LIN {X 0,Y 291.334,Z 480.193,A -85,B 0,C 180,E1 -16780.643,E2 -16780.643} C_VEL
LIN {X 0,Y 291.294,Z 480.201,A -85,B 0,C 180,E1 -16784.402,E2 -16784.402} C_VEL
LIN {X 0,Y 291.33,Z 480.196,A -85,B 0,C 180,E1 -16788.405,E2 -16788.405} C_VEL
LIN {X 0,Y 291.368,Z 480.187,A -85,B 0,C 180,E1 -16791.161,E2 -16791.161} C_VEL
LIN {X 0,Y 291.389,Z 480.187,A -85,B 0,C 180,E1 -16794.63,E2 -16794.63} C_VEL
LIN {X 0,Y 291.377,Z 480.19,A -85,B 0,C 180,E1 -16797.951,E2 -16797.951} C_VEL
LIN {X 0,Y 291.386,Z 480.185,A -85,B 0,C 180,E1 -16801.159,E2 -16801.159} C_VEL
LIN {X 0,Y 291.422,Z 480.185,A -85,B 0,C 180,E1 -16804.272,E2 -16804.272} C_VEL
LIN {X 0,Y 291.386,Z 480.185,A -85,B 0,C 180,E1 -16807.3,E2 -16807.3} C_VEL
LIN {X 0,Y 291.463,Z 480.18,A -85,B 0,C 180,E1 -16810.27,E2 -16810.27} C_VEL
LIN {X 0,Y 291.56,Z 480.165,A -85,B 0,C 180,E1 -16814.624,E2 -16814.624} C_VEL
LIN {X 0,Y 291.542,Z 480.166,A -85,B 0,C 180,E1 -16818.881,E2 -16818.881} C_VEL
LIN {X 0,Y 291.714,Z 480.147,A -85,B 0,C 180,E1 -16821.689,E2 -16821.689} C_VEL
LIN {X 0,Y 291.635,Z 480.156,A -85,B 0,C 180,E1 -16824.468,E2 -16824.468} C_VEL
LIN {X 0,Y 291.893,Z 480.123,A -85,B 0,C 180,E1 -16828.62,E2 -16828.62} C_VEL
LIN {X 0,Y 291.893,Z 480.123,A -85,B 0,C 180,E1 -16831.38,E2 -16831.38} C_VEL
LIN {X 0,Y 291.616,Z 480.158,A -85,B 0,C 180,E1 -16835.532,E2 -16835.532} C_VEL
LIN {X 0,Y 291.678,Z 480.149,A -85,B 0,C 180,E1 -16838.919,E2 -16838.919} C_VEL
LIN {X 0,Y 291.525,Z 480.168,A -85,B 0,C 180,E1 -16842.531,E2 -16842.531} C_VEL
LIN {X 0,Y 291.56,Z 480.165,A -85,B 0,C 180,E1 -16845.376,E2 -16845.376} C_VEL
LIN {X 0,Y 291.455,Z 480.182,A -85,B 0,C 180,E1 -16849.875,E2 -16849.875} C_VEL
LIN {X 0,Y 291.403,Z 480.186,A -85,B 0,C 180,E1 -16854.205,E2 -16854.205} C_VEL
LIN {X 0,Y 291.424,Z 480.182,A -85,B 0,C 180,E1 -16857.272,E2 -16857.272} C_VEL
LIN {X 0,Y 291.338,Z 480.191,A -85,B 0,C 180,E1 -16860.437,E2 -16860.437} C_VEL
LIN {X 0,Y 291.349,Z 480.194,A -85,B 0,C 180,E1 -16863.698,E2 -16863.698} C_VEL
LIN {X 0,Y 291.398,Z 480.185,A -85,B 0,C 180,E1 -16867.259,E2 -16867.259} C_VEL
LIN {X 0,Y 291.338,Z 480.191,A -85,B 0,C 180,E1 -16870.642,E2 -16870.642} C_VEL
LIN {X 0,Y 291.293,Z 480.198,A -85,B 0,C 180,E1 -16874.402,E2 -16874.402} C_VEL
LIN {X 0,Y 291.329,Z 480.192,A -85,B 0,C 180,E1 -16878.404,E2 -16878.404} C_VEL
LIN {X 0,Y 291.347,Z 480.192,A -85,B 0,C 180,E1 -16881.157,E2 -16881.157} C_VEL
LIN {X 0,Y 291.375,Z 480.187,A -85,B 0,C 180,E1 -16882.914,E2 -16882.914} C_VEL
LIN {X 0,Y 291.126,Z 480.218,A -85,B 0,C 180,E1 -16886.272,E2 -16886.272} C_VEL
LIN {X 0,Y 290.796,Z 480.263,A -85,B 0,C 180,E1 -16889.5,E2 -16889.5} C_VEL
LIN {X 0,Y 290.411,Z 480.307,A -85,B 0,C 180,E1 -16892.625,E2 -16892.625} C_VEL
LIN {X 0,Y 289.943,Z 480.417,A -85,B 0,C 180,E1 -16896.236,E2 -16896.236} C_VEL
LIN {X 0,Y 289.946,Z 482.927,A -85,B 0,C 180,E1 -16898.679,E2 -16898.679} C_VEL
LIN {X 0,Y 292.691,Z 498.006,A -85,B 0,C 180,E1 -16899.711,E2 -16899.711} C_VEL
LIN {X 0,Y 295.355,Z 512.188,A -85,B 0,C 180,E1 -16900.992,E2 -16900.992} C_VEL
LIN {X 0,Y 295.583,Z 516.745,A -85,B 0,C 180,E1 -16901.457,E2 -16901.457} C_VEL
LIN {X 0,Y 294.542,Z 528.4,A -85,B 0,C 180,E1 -16902.788,E2 -16902.788} C_VEL
LIN {X 0,Y 293.546,Z 538.437,A -85,B 0,C 180,E1 -16904.196,E2 -16904.196} C_VEL
LIN {X 0,Y 292.641,Z 547.665,A -85,B 0,C 180,E1 -16905.749,E2 -16905.749} C_VEL
LIN {X 0,Y 291.737,Z 556.266,A -85,B 0,C 180,E1 -16907.478,E2 -16907.478} C_VEL
LIN {X 0,Y 290.974,Z 564.767,A -85,B 0,C 180,E1 -16909.563,E2 -16909.563} C_VEL
LIN {X 0,Y 290.377,Z 571.664,A -85,B 0,C 180,E1 -16911.65,E2 -16911.65} C_VEL
LIN {X 0,Y 290.067,Z 576.41,A -85,B 0,C 180,E1 -16913.408,E2 -16913.408} C_VEL
LIN {X 0,Y 289.833,Z 581.565,A -85,B 0,C 180,E1 -16915.828,E2 -16915.828} C_VEL
LIN {X 0,Y 289.714,Z 583.883,A -85,B 0,C 180,E1 -16917.219,E2 -16917.219} C_VEL
LIN {X 0,Y 289.64,Z 585.506,A -85,B 0,C 180,E1 -16918.442,E2 -16918.442} C_VEL
LIN {X 0,Y 289.01,Z 586.88,A -85,B 0,C 180,E1 -16919.573,E2 -16919.573} C_VEL
LIN {X 0,Y 286.338,Z 588.547,A -85,B 0,C 180,E1 -16921.444,E2 -16921.444} C_VEL
LIN {X 0,Y 284.137,Z 589.296,A -85,B 0,C 180,E1 -16922.979,E2 -16922.979} C_VEL
LIN {X 0,Y 283.277,Z 589.509,A -85,B 0,C 180,E1 -16924.167,E2 -16924.167} C_VEL
LIN {X 0,Y 283.251,Z 589.501,A -85,B 0,C 180,E1 -16924.568,E2 -16924.568} C_VEL
LIN {X 0,Y 283.807,Z 588.988,A -85,B 0,C 180,E1 -16927.112,E2 -16927.112} C_VEL
LIN {X 0,Y 285.067,Z 587.261,A -85,B 0,C 180,E1 -16929.544,E2 -16929.544} C_VEL
LIN {X 0,Y 286.508,Z 584.256,A -85,B 0,C 180,E1 -16932.034,E2 -16932.034} C_VEL
LIN {X 0,Y 288.806,Z 579.257,A -85,B 0,C 180,E1 -16934.804,E2 -16934.804} C_VEL
LIN {X 0,Y 290.955,Z 574.336,A -85,B 0,C 180,E1 -16936.849,E2 -16936.849} C_VEL
LIN {X 0,Y 293.872,Z 567.073,A -85,B 0,C 180,E1 -16939.198,E2 -16939.198} C_VEL
LIN {X 0,Y 296.873,Z 559.452,A -85,B 0,C 180,E1 -16941.163,E2 -16941.163} C_VEL
LIN {X 0,Y 300.223,Z 550.179,A -85,B 0,C 180,E1 -16943.085,E2 -16943.085} C_VEL
LIN {X 0,Y 303.614,Z 539.794,A -85,B 0,C 180,E1 -16944.831,E2 -16944.831} C_VEL
LIN {X 0,Y 304.404,Z 537.308,A -85,B 0,C 180,E1 -16945.191,E2 -16945.191} C_VEL
LIN {X 0,Y 304.646,Z 535.637,A -85,B 0,C 180,E1 -16945.489,E2 -16945.489} C_VEL
LIN {X 0,Y 303.451,Z 527.808,A -85,B 0,C 180,E1 -16947.303,E2 -16947.303} C_VEL
LIN {X 0,Y 301.243,Z 520.052,A -85,B 0,C 180,E1 -16949.336,E2 -16949.336} C_VEL
LIN {X 0,Y 298.599,Z 513.072,A -85,B 0,C 180,E1 -16951.459,E2 -16951.459} C_VEL
LIN {X 0,Y 296.624,Z 508.611,A -85,B 0,C 180,E1 -16953.021,E2 -16953.021} C_VEL
LIN {X 0,Y 294.159,Z 504.223,A -85,B 0,C 180,E1 -16954.988,E2 -16954.988} C_VEL
LIN {X 0,Y 291.916,Z 500.866,A -85,B 0,C 180,E1 -16957.005,E2 -16957.005} C_VEL
LIN {X 0,Y 291.673,Z 500.148,A -85,B 0,C 180,E1 -16957.33,E2 -16957.33} C_VEL
LIN {X 0,Y 288.682,Z 497.206,A -85,B 0,C 180,E1 -16961.096,E2 -16961.096} C_VEL
LIN {X 0,Y 288.16,Z 496.183,A -85,B 0,C 180,E1 -16963.31,E2 -16963.31} C_VEL
LIN {X 0,Y 288.331,Z 496.661,A -85,B 0,C 180,E1 -16965.019,E2 -16965.019} C_VEL
LIN {X 0,Y 288.629,Z 498.198,A -85,B 0,C 180,E1 -16967.855,E2 -16967.855} C_VEL
LIN {X 0,Y 290.515,Z 502.885,A -85,B 0,C 180,E1 -16971.025,E2 -16971.025} C_VEL
LIN {X 0,Y 292.089,Z 505.556,A -85,B 0,C 180,E1 -16972.563,E2 -16972.563} C_VEL
LIN {X 0,Y 294.502,Z 513.126,A -85,B 0,C 180,E1 -16975.059,E2 -16975.059} C_VEL
LIN {X 0,Y 296.539,Z 520.344,A -85,B 0,C 180,E1 -16976.968,E2 -16976.968} C_VEL
LIN {X 0,Y 297.747,Z 527.635,A -85,B 0,C 180,E1 -16978.485,E2 -16978.485} C_VEL
LIN {X 0,Y 299.033,Z 539.159,A -85,B 0,C 180,E1 -16980.658,E2 -16980.658} C_VEL
LIN {X 0,Y 299.343,Z 551.45,A -85,B 0,C 180,E1 -16982.829,E2 -16982.829} C_VEL
LIN {X 0,Y 298.611,Z 562.364,A -85,B 0,C 180,E1 -16984.739,E2 -16984.739} C_VEL
LIN {X 0,Y 296.615,Z 572.882,A -85,B 0,C 180,E1 -16986.617,E2 -16986.617} C_VEL
LIN {X 0,Y 293.295,Z 582.962,A -85,B 0,C 180,E1 -16988.566,E2 -16988.566} C_VEL
LIN {X 0,Y 290.399,Z 591.537,A -85,B 0,C 180,E1 -16990.609,E2 -16990.609} C_VEL
LIN {X 0,Y 288.013,Z 598.477,A -85,B 0,C 180,E1 -16992.607,E2 -16992.607} C_VEL
LIN {X 0,Y 285.907,Z 605.175,A -85,B 0,C 180,E1 -16995.042,E2 -16995.042} C_VEL
LIN {X 0,Y 284.328,Z 609.813,A -85,B 0,C 180,E1 -16997.146,E2 -16997.146} C_VEL
LIN {X 0,Y 283.152,Z 614.446,A -85,B 0,C 180,E1 -16999.994,E2 -16999.994} C_VEL
LIN {X 0,Y 282.803,Z 616.163,A -85,B 0,C 180,E1 -17001.425,E2 -17001.425} C_VEL
LIN {X 0,Y 282.522,Z 618.348,A -85,B 0,C 180,E1 -17004.289,E2 -17004.289} C_VEL
LIN {X 0,Y 282.52,Z 618.859,A -85,B 0,C 180,E1 -17005.72,E2 -17005.72} C_VEL
LIN {X 0,Y 282.582,Z 618.969,A -85,B 0,C 180,E1 -17007.149,E2 -17007.149} C_VEL
LIN {X 0,Y 282.866,Z 618.592,A -85,B 0,C 180,E1 -17008.932,E2 -17008.932} C_VEL
LIN {X 0,Y 282.885,Z 619.433,A -85,B 0,C 180,E1 -17010,E2 -17010} C_VEL
LIN {X 0,Y 282.703,Z 620.169,A -85,B 0,C 180,E1 -17011.425,E2 -17011.425} C_VEL
LIN {X 0,Y 282.498,Z 620.489,A -85,B 0,C 180,E1 -17012.852,E2 -17012.852} C_VEL
LIN {X 0,Y 282.442,Z 619.945,A -85,B 0,C 180,E1 -17015.546,E2 -17015.546} C_VEL
LIN {X 0,Y 282.549,Z 618.968,A -85,B 0,C 180,E1 -17017.144,E2 -17017.144} C_VEL
LIN {X 0,Y 282.796,Z 617.689,A -85,B 0,C 180,E1 -17018.575,E2 -17018.575} C_VEL
LIN {X 0,Y 283.705,Z 613.888,A -85,B 0,C 180,E1 -17021.43,E2 -17021.43} C_VEL
LIN {X 0,Y 284.793,Z 609.991,A -85,B 0,C 180,E1 -17023.558,E2 -17023.558} C_VEL
LIN {X 0,Y 286.466,Z 605.074,A -85,B 0,C 180,E1 -17025.656,E2 -17025.656} C_VEL
LIN {X 0,Y 289.04,Z 596.909,A -85,B 0,C 180,E1 -17028.427,E2 -17028.427} C_VEL
LIN {X 0,Y 292.268,Z 587.863,A -85,B 0,C 180,E1 -17030.774,E2 -17030.774} C_VEL
LIN {X 0,Y 295.55,Z 578.572,A -85,B 0,C 180,E1 -17032.732,E2 -17032.732} C_VEL
LIN {X 0,Y 297.766,Z 571.418,A -85,B 0,C 180,E1 -17034.025,E2 -17034.025} C_VEL
LIN {X 0,Y 299.353,Z 562.829,A -85,B 0,C 180,E1 -17035.534,E2 -17035.534} C_VEL
LIN {X 0,Y 299.795,Z 553.607,A -85,B 0,C 180,E1 -17037.202,E2 -17037.202} C_VEL
LIN {X 0,Y 299.141,Z 543.023,A -85,B 0,C 180,E1 -17039.207,E2 -17039.207} C_VEL
LIN {X 0,Y 297.549,Z 532.972,A -85,B 0,C 180,E1 -17041.308,E2 -17041.308} C_VEL
LIN {X 0,Y 295.334,Z 523.354,A -85,B 0,C 180,E1 -17043.603,E2 -17043.603} C_VEL
LIN {X 0,Y 293.444,Z 516.852,A -85,B 0,C 180,E1 -17045.482,E2 -17045.482} C_VEL
LIN {X 0,Y 292.016,Z 512.481,A -85,B 0,C 180,E1 -17046.99,E2 -17046.99} C_VEL
LIN {X 0,Y 291.808,Z 511.167,A -85,B 0,C 180,E1 -17047.365,E2 -17047.365} C_VEL
LIN {X 0,Y 288.758,Z 504.957,A -85,B 0,C 180,E1 -17051.083,E2 -17051.083} C_VEL
LIN {X 0,Y 288.003,Z 501.761,A -85,B 0,C 180,E1 -17053.544,E2 -17053.544} C_VEL
LIN {X 0,Y 287.807,Z 500.618,A -85,B 0,C 180,E1 -17055.975,E2 -17055.975} C_VEL
LIN {X 0,Y 288.439,Z 501.626,A -85,B 0,C 180,E1 -17059.055,E2 -17059.055} C_VEL
LIN {X 0,Y 291.413,Z 503.824,A -85,B 0,C 180,E1 -17062.737,E2 -17062.737} C_VEL
LIN {X 0,Y 292.328,Z 505.916,A -85,B 0,C 180,E1 -17063.863,E2 -17063.863} C_VEL
LIN {X 0,Y 293.661,Z 507.267,A -85,B 0,C 180,E1 -17064.944,E2 -17064.944} C_VEL
LIN {X 0,Y 296.553,Z 512.135,A -85,B 0,C 180,E1 -17067.281,E2 -17067.281} C_VEL
LIN {X 0,Y 300.148,Z 519.88,A -85,B 0,C 180,E1 -17070.039,E2 -17070.039} C_VEL
LIN {X 0,Y 302.846,Z 527.891,A -85,B 0,C 180,E1 -17072.346,E2 -17072.346} C_VEL
LIN {X 0,Y 304.613,Z 536.548,A -85,B 0,C 180,E1 -17074.514,E2 -17074.514} C_VEL
LIN {X 0,Y 304.698,Z 537.826,A -85,B 0,C 180,E1 -17074.798,E2 -17074.798} C_VEL
LIN {X 0,Y 301.105,Z 548.999,A -85,B 0,C 180,E1 -17076.622,E2 -17076.622} C_VEL
LIN {X 0,Y 297.665,Z 558.567,A -85,B 0,C 180,E1 -17078.533,E2 -17078.533} C_VEL
LIN {X 0,Y 294.039,Z 567.574,A -85,B 0,C 180,E1 -17080.814,E2 -17080.814} C_VEL
LIN {X 0,Y 291.091,Z 574.794,A -85,B 0,C 180,E1 -17083.159,E2 -17083.159} C_VEL
LIN {X 0,Y 288.974,Z 579.689,A -85,B 0,C 180,E1 -17085.205,E2 -17085.205} C_VEL
LIN {X 0,Y 286.607,Z 584.705,A -85,B 0,C 180,E1 -17087.97,E2 -17087.97} C_VEL
LIN {X 0,Y 285.258,Z 587.491,A -85,B 0,C 180,E1 -17090.231,E2 -17090.231} C_VEL
LIN {X 0,Y 283.867,Z 589.466,A -85,B 0,C 180,E1 -17092.889,E2 -17092.889} C_VEL
LIN {X 0,Y 283.578,Z 589.924,A -85,B 0,C 180,E1 -17094.311,E2 -17094.311} C_VEL
LIN {X 0,Y 283.299,Z 590.016,A -85,B 0,C 180,E1 -17095.732,E2 -17095.732} C_VEL
LIN {X 0,Y 282.979,Z 589.737,A -85,B 0,C 180,E1 -17097.153,E2 -17097.153} C_VEL
LIN {X 0,Y 282.754,Z 589.038,A -85,B 0,C 180,E1 -17098.576,E2 -17098.576} C_VEL
LIN {X 0,Y 282.586,Z 586.427,A -85,B 0,C 180,E1 -17101.425,E2 -17101.425} C_VEL
LIN {X 0,Y 282.709,Z 583.358,A -85,B 0,C 180,E1 -17103.564,E2 -17103.564} C_VEL
LIN {X 0,Y 282.844,Z 579.26,A -85,B 0,C 180,E1 -17105.704,E2 -17105.704} C_VEL
LIN {X 0,Y 283.281,Z 573.055,A -85,B 0,C 180,E1 -17108.202,E2 -17108.202} C_VEL
LIN {X 0,Y 283.949,Z 565.036,A -85,B 0,C 180,E1 -17110.698,E2 -17110.698} C_VEL
LIN {X 0,Y 284.75,Z 556.478,A -85,B 0,C 180,E1 -17112.835,E2 -17112.835} C_VEL
LIN {X 0,Y 285.914,Z 545.866,A -85,B 0,C 180,E1 -17114.958,E2 -17114.958} C_VEL
LIN {X 0,Y 287.022,Z 536.197,A -85,B 0,C 180,E1 -17116.538,E2 -17116.538} C_VEL
LIN {X 0,Y 287.925,Z 525.259,A -85,B 0,C 180,E1 -17118.012,E2 -17118.012} C_VEL
LIN {X 0,Y 288.683,Z 516.455,A -85,B 0,C 180,E1 -17119.003,E2 -17119.003} C_VEL
LIN {X 0,Y 288.131,Z 511.699,A -85,B 0,C 180,E1 -17119.504,E2 -17119.504} C_VEL
LIN {X 0,Y 285.556,Z 498.301,A -85,B 0,C 180,E1 -17120.732,E2 -17120.732} C_VEL
LIN {X 0,Y 282.979,Z 484.536,A -85,B 0,C 180,E1 -17121.705,E2 -17121.705} C_VEL
LIN {X 0,Y 282.92,Z 484.131,A -85,B 0,C 180,E1 -17121.756,E2 -17121.756} C_VEL
LIN {X 0,Y 283.028,Z 481.339,A -85,B 0,C 180,E1 -17124.97,E2 -17124.97} C_VEL
LIN {X 0,Y 283.396,Z 481.187,A -85,B 0,C 180,E1 -17128.112,E2 -17128.112} C_VEL
LIN {X 0,Y 283.732,Z 481.139,A -85,B 0,C 180,E1 -17131.344,E2 -17131.344} C_VEL
LIN {X 0,Y 284.129,Z 481.09,A -85,B 0,C 180,E1 -17135.287,E2 -17135.287} C_VEL
LIN {X 0,Y 284.269,Z 481.077,A -85,B 0,C 180,E1 -17138.176,E2 -17138.176} C_VEL
LIN {X 0,Y 284.275,Z 481.072,A -85,B 0,C 180,E1 -17141.876,E2 -17141.876} C_VEL
LIN {X 0,Y 284.259,Z 481.078,A -85,B 0,C 180,E1 -17146.19,E2 -17146.19} C_VEL
LIN {X 0,Y 284.31,Z 481.07,A -85,B 0,C 180,E1 -17150.024,E2 -17150.024} C_VEL
LIN {X 0,Y 284.354,Z 481.063,A -85,B 0,C 180,E1 -17153.617,E2 -17153.617} C_VEL
LIN {X 0,Y 284.312,Z 481.067,A -85,B 0,C 180,E1 -17157.19,E2 -17157.19} C_VEL
LIN {X 0,Y 284.363,Z 481.064,A -85,B 0,C 180,E1 -17160.376,E2 -17160.376} C_VEL
LIN {X 0,Y 284.382,Z 481.059,A -85,B 0,C 180,E1 -17163.587,E2 -17163.587} C_VEL
LIN {X 0,Y 284.371,Z 481.06,A -85,B 0,C 180,E1 -17166.707,E2 -17166.707} C_VEL
LIN {X 0,Y 284.408,Z 481.055,A -85,B 0,C 180,E1 -17171.262,E2 -17171.262} C_VEL
LIN {X 0,Y 284.497,Z 481.046,A -85,B 0,C 180,E1 -17174.459,E2 -17174.459} C_VEL
LIN {X 0,Y 284.493,Z 481.045,A -85,B 0,C 180,E1 -17178.602,E2 -17178.602} C_VEL
LIN {X 0,Y 284.664,Z 481.024,A -85,B 0,C 180,E1 -17181.481,E2 -17181.481} C_VEL
LIN {X 0,Y 284.606,Z 481.032,A -85,B 0,C 180,E1 -17184.331,E2 -17184.331} C_VEL
LIN {X 0,Y 284.859,Z 481,A -85,B 0,C 180,E1 -17188.586,E2 -17188.586} C_VEL
LIN {X 0,Y 284.859,Z 481,A -85,B 0,C 180,E1 -17191.414,E2 -17191.414} C_VEL
LIN {X 0,Y 284.658,Z 481.024,A -85,B 0,C 180,E1 -17197.091,E2 -17197.091} C_VEL
LIN {X 0,Y 284.522,Z 481.046,A -85,B 0,C 180,E1 -17199.957,E2 -17199.957} C_VEL
LIN {X 0,Y 284.486,Z 481.047,A -85,B 0,C 180,E1 -17204.303,E2 -17204.303} C_VEL
LIN {X 0,Y 284.43,Z 481.053,A -85,B 0,C 180,E1 -17207.248,E2 -17207.248} C_VEL
LIN {X 0,Y 284.382,Z 481.06,A -85,B 0,C 180,E1 -17210.242,E2 -17210.242} C_VEL
LIN {X 0,Y 284.371,Z 481.064,A -85,B 0,C 180,E1 -17213.874,E2 -17213.874} C_VEL
LIN {X 0,Y 284.399,Z 481.057,A -85,B 0,C 180,E1 -17217.173,E2 -17217.173} C_VEL
LIN {X 0,Y 284.298,Z 481.068,A -85,B 0,C 180,E1 -17221.274,E2 -17221.274} C_VEL
LIN {X 0,Y 284.366,Z 481.062,A -85,B 0,C 180,E1 -17225.354,E2 -17225.354} C_VEL
LIN {X 0,Y 284.327,Z 481.066,A -85,B 0,C 180,E1 -17228.167,E2 -17228.167} C_VEL
LIN {X 0,Y 284.273,Z 481.074,A -85,B 0,C 180,E1 -17232.124,E2 -17232.124} C_VEL
LIN {X 0,Y 284.258,Z 481.075,A -85,B 0,C 180,E1 -17236.189,E2 -17236.189} C_VEL
LIN {X 0,Y 284.309,Z 481.07,A -85,B 0,C 180,E1 -17240.024,E2 -17240.024} C_VEL
LIN {X 0,Y 284.254,Z 481.079,A -85,B 0,C 180,E1 -17243.602,E2 -17243.602} C_VEL
LIN {X 0,Y 283.996,Z 481.107,A -85,B 0,C 180,E1 -17247.288,E2 -17247.288} C_VEL
LIN {X 0,Y 283.674,Z 481.147,A -85,B 0,C 180,E1 -17250.297,E2 -17250.297} C_VEL
LIN {X 0,Y 283.27,Z 481.2,A -85,B 0,C 180,E1 -17253.475,E2 -17253.475} C_VEL
LIN {X 0,Y 282.87,Z 481.398,A -85,B 0,C 180,E1 -17256.576,E2 -17256.576} C_VEL
LIN {X 0,Y 282.863,Z 483.281,A -85,B 0,C 180,E1 -17258.43,E2 -17258.43} C_VEL
LIN {X 0,Y 285.601,Z 498.484,A -85,B 0,C 180,E1 -17259.494,E2 -17259.494} C_VEL
LIN {X 0,Y 288.16,Z 512.297,A -85,B 0,C 180,E1 -17260.776,E2 -17260.776} C_VEL
LIN {X 0,Y 288.606,Z 516.076,A -85,B 0,C 180,E1 -17261.176,E2 -17261.176} C_VEL
LIN {X 0,Y 287.539,Z 528.127,A -85,B 0,C 180,E1 -17262.561,E2 -17262.561} C_VEL
LIN {X 0,Y 286.543,Z 538.135,A -85,B 0,C 180,E1 -17263.982,E2 -17263.982} C_VEL
LIN {X 0,Y 285.508,Z 548.416,A -85,B 0,C 180,E1 -17265.749,E2 -17265.749} C_VEL
LIN {X 0,Y 284.62,Z 556.944,A -85,B 0,C 180,E1 -17267.522,E2 -17267.522} C_VEL
LIN {X 0,Y 283.836,Z 565.352,A -85,B 0,C 180,E1 -17269.658,E2 -17269.658} C_VEL
LIN {X 0,Y 283.164,Z 573.225,A -85,B 0,C 180,E1 -17272.154,E2 -17272.154} C_VEL
LIN {X 0,Y 282.822,Z 578.538,A -85,B 0,C 180,E1 -17274.295,E2 -17274.295} C_VEL
LIN {X 0,Y 282.704,Z 582.701,A -85,B 0,C 180,E1 -17276.436,E2 -17276.436} C_VEL
LIN {X 0,Y 282.556,Z 585.827,A -85,B 0,C 180,E1 -17278.574,E2 -17278.574} C_VEL
LIN {X 0,Y 282.585,Z 587.35,A -85,B 0,C 180,E1 -17280,E2 -17280} C_VEL
LIN {X 0,Y 282.959,Z 589.213,A -85,B 0,C 180,E1 -17282.847,E2 -17282.847} C_VEL
LIN {X 0,Y 283.251,Z 589.501,A -85,B 0,C 180,E1 -17284.568,E2 -17284.568} C_VEL
LIN {X 0,Y 282.838,Z 589.496,A -85,B 0,C 180,E1 -17285.762,E2 -17285.762} C_VEL
LIN {X 0,Y 280.687,Z 589.079,A -85,B 0,C 180,E1 -17287.728,E2 -17287.728} C_VEL
LIN {X 0,Y 279.018,Z 588.352,A -85,B 0,C 180,E1 -17289.312,E2 -17289.312} C_VEL
LIN {X 0,Y 278.595,Z 587.463,A -85,B 0,C 180,E1 -17290.51,E2 -17290.51} C_VEL
LIN {X 0,Y 278.718,Z 587.033,A -85,B 0,C 180,E1 -17290.907,E2 -17290.907} C_VEL
LIN {X 0,Y 280.844,Z 583.239,A -85,B 0,C 180,E1 -17293.753,E2 -17293.753} C_VEL
LIN {X 0,Y 282.762,Z 579.256,A -85,B 0,C 180,E1 -17295.867,E2 -17295.867} C_VEL
LIN {X 0,Y 286.063,Z 572.265,A -85,B 0,C 180,E1 -17298.625,E2 -17298.625} C_VEL
LIN {X 0,Y 288.947,Z 565.685,A -85,B 0,C 180,E1 -17300.651,E2 -17300.651} C_VEL
LIN {X 0,Y 292.892,Z 556.155,A -85,B 0,C 180,E1 -17302.949,E2 -17302.949} C_VEL
LIN {X 0,Y 296.576,Z 546.223,A -85,B 0,C 180,E1 -17304.874,E2 -17304.874} C_VEL
LIN {X 0,Y 299.027,Z 538.923,A -85,B 0,C 180,E1 -17306.052,E2 -17306.052} C_VEL
LIN {X 0,Y 298.223,Z 531.607,A -85,B 0,C 180,E1 -17307.886,E2 -17307.886} C_VEL
LIN {X 0,Y 296.52,Z 524.617,A -85,B 0,C 180,E1 -17309.85,E2 -17309.85} C_VEL
LIN {X 0,Y 294.334,Z 518.114,A -85,B 0,C 180,E1 -17311.968,E2 -17311.968} C_VEL
LIN {X 0,Y 292.69,Z 514.063,A -85,B 0,C 180,E1 -17313.523,E2 -17313.523} C_VEL
LIN {X 0,Y 290.6,Z 510.045,A -85,B 0,C 180,E1 -17315.48,E2 -17315.48} C_VEL
LIN {X 0,Y 288.817,Z 506.78,A -85,B 0,C 180,E1 -17317.47,E2 -17317.47} C_VEL
LIN {X 0,Y 286.562,Z 504.367,A -85,B 0,C 180,E1 -17320.511,E2 -17320.511} C_VEL
LIN {X 0,Y 285.897,Z 503.169,A -85,B 0,C 180,E1 -17322.484,E2 -17322.484} C_VEL
LIN {X 0,Y 285.76,Z 502.894,A -85,B 0,C 180,E1 -17323.522,E2 -17323.522} C_VEL
LIN {X 0,Y 285.852,Z 503.946,A -85,B 0,C 180,E1 -17326.495,E2 -17326.495} C_VEL
LIN {X 0,Y 286.181,Z 504.586,A -85,B 0,C 180,E1 -17327.454,E2 -17327.454} C_VEL
LIN {X 0,Y 286.938,Z 507.161,A -85,B 0,C 180,E1 -17329.401,E2 -17329.401} C_VEL
LIN {X 0,Y 289.078,Z 511.633,A -85,B 0,C 180,E1 -17332.151,E2 -17332.151} C_VEL
LIN {X 0,Y 290.887,Z 518.691,A -85,B 0,C 180,E1 -17334.56,E2 -17334.56} C_VEL
LIN {X 0,Y 292.401,Z 525.501,A -85,B 0,C 180,E1 -17336.439,E2 -17336.439} C_VEL
LIN {X 0,Y 293.306,Z 533.543,A -85,B 0,C 180,E1 -17338.187,E2 -17338.187} C_VEL
LIN {X 0,Y 293.907,Z 545.279,A -85,B 0,C 180,E1 -17340.514,E2 -17340.514} C_VEL
LIN {X 0,Y 293.543,Z 556.422,A -85,B 0,C 180,E1 -17342.602,E2 -17342.602} C_VEL
LIN {X 0,Y 292.673,Z 564.547,A -85,B 0,C 180,E1 -17344.12,E2 -17344.12} C_VEL
LIN {X 0,Y 290.317,Z 574.843,A -85,B 0,C 180,E1 -17346.078,E2 -17346.078} C_VEL
LIN {X 0,Y 286.831,Z 584.441,A -85,B 0,C 180,E1 -17348.058,E2 -17348.058} C_VEL
LIN {X 0,Y 283.275,Z 593.972,A -85,B 0,C 180,E1 -17350.523,E2 -17350.523} C_VEL
LIN {X 0,Y 280.949,Z 600.21,A -85,B 0,C 180,E1 -17352.531,E2 -17352.531} C_VEL
LIN {X 0,Y 279.083,Z 605.643,A -85,B 0,C 180,E1 -17354.668,E2 -17354.668} C_VEL
LIN {X 0,Y 277.394,Z 610.038,A -85,B 0,C 180,E1 -17356.819,E2 -17356.819} C_VEL
LIN {X 0,Y 276.707,Z 612.448,A -85,B 0,C 180,E1 -17358.276,E2 -17358.276} C_VEL
LIN {X 0,Y 276.144,Z 614.435,A -85,B 0,C 180,E1 -17359.738,E2 -17359.738} C_VEL
LIN {X 0,Y 275.519,Z 617.203,A -85,B 0,C 180,E1 -17362.672,E2 -17362.672} C_VEL
LIN {X 0,Y 275.427,Z 618.113,A -85,B 0,C 180,E1 -17364.356,E2 -17364.356} C_VEL
LIN {X 0,Y 275.501,Z 618.403,A -85,B 0,C 180,E1 -17367.076,E2 -17367.076} C_VEL
LIN {X 0,Y 275.807,Z 617.967,A -85,B 0,C 180,E1 -17369.087,E2 -17369.087} C_VEL
LIN {X 0,Y 275.832,Z 618.719,A -85,B 0,C 180,E1 -17370,E2 -17370} C_VEL
LIN {X 0,Y 275.635,Z 619.518,A -85,B 0,C 180,E1 -17371.461,E2 -17371.461} C_VEL
LIN {X 0,Y 275.385,Z 619.928,A -85,B 0,C 180,E1 -17374.391,E2 -17374.391} C_VEL
LIN {X 0,Y 275.375,Z 619.518,A -85,B 0,C 180,E1 -17375.859,E2 -17375.859} C_VEL
LIN {X 0,Y 275.737,Z 617.51,A -85,B 0,C 180,E1 -17378.797,E2 -17378.797} C_VEL
LIN {X 0,Y 276.725,Z 613.993,A -85,B 0,C 180,E1 -17381.723,E2 -17381.723} C_VEL
LIN {X 0,Y 277.891,Z 610.252,A -85,B 0,C 180,E1 -17383.902,E2 -17383.902} C_VEL
LIN {X 0,Y 279.649,Z 605.583,A -85,B 0,C 180,E1 -17386.048,E2 -17386.048} C_VEL
LIN {X 0,Y 281.978,Z 598.92,A -85,B 0,C 180,E1 -17388.502,E2 -17388.502} C_VEL
LIN {X 0,Y 285.226,Z 590.488,A -85,B 0,C 180,E1 -17390.933,E2 -17390.933} C_VEL
LIN {X 0,Y 288.562,Z 581.857,A -85,B 0,C 180,E1 -17392.935,E2 -17392.935} C_VEL
LIN {X 0,Y 291.546,Z 573.459,A -85,B 0,C 180,E1 -17394.572,E2 -17394.572} C_VEL
LIN {X 0,Y 293.475,Z 564.757,A -85,B 0,C 180,E1 -17396.203,E2 -17396.203} C_VEL
LIN {X 0,Y 294.102,Z 556.252,A -85,B 0,C 180,E1 -17397.851,E2 -17397.851} C_VEL
LIN {X 0,Y 293.845,Z 546.614,A -85,B 0,C 180,E1 -17399.802,E2 -17399.802} C_VEL
LIN {X 0,Y 292.767,Z 537.312,A -85,B 0,C 180,E1 -17401.879,E2 -17401.879} C_VEL
LIN {X 0,Y 291.145,Z 528.37,A -85,B 0,C 180,E1 -17404.153,E2 -17404.153} C_VEL
LIN {X 0,Y 289.65,Z 522.168,A -85,B 0,C 180,E1 -17406.048,E2 -17406.048} C_VEL
LIN {X 0,Y 288.232,Z 516.629,A -85,B 0,C 180,E1 -17408.07,E2 -17408.07} C_VEL
LIN {X 0,Y 285.927,Z 511.034,A -85,B 0,C 180,E1 -17411.579,E2 -17411.579} C_VEL
LIN {X 0,Y 285.481,Z 508.502,A -85,B 0,C 180,E1 -17413.575,E2 -17413.575} C_VEL
LIN {X 0,Y 285.312,Z 507.375,A -85,B 0,C 180,E1 -17415.59,E2 -17415.59} C_VEL
LIN {X 0,Y 285.432,Z 507.656,A -85,B 0,C 180,E1 -17417.618,E2 -17417.618} C_VEL
LIN {X 0,Y 287.387,Z 509.554,A -85,B 0,C 180,E1 -17421.495,E2 -17421.495} C_VEL
LIN {X 0,Y 288.349,Z 510.171,A -85,B 0,C 180,E1 -17422.459,E2 -17422.459} C_VEL
LIN {X 0,Y 288.914,Z 511.737,A -85,B 0,C 180,E1 -17423.393,E2 -17423.393} C_VEL
LIN {X 0,Y 290.839,Z 514.424,A -85,B 0,C 180,E1 -17425.245,E2 -17425.245} C_VEL
LIN {X 0,Y 293.416,Z 519.69,A -85,B 0,C 180,E1 -17427.671,E2 -17427.671} C_VEL
LIN {X 0,Y 295.569,Z 524.835,A -85,B 0,C 180,E1 -17429.612,E2 -17429.612} C_VEL
LIN {X 0,Y 297.986,Z 533.332,A -85,B 0,C 180,E1 -17432.203,E2 -17432.203} C_VEL
LIN {X 0,Y 298.981,Z 539.528,A -85,B 0,C 180,E1 -17433.87,E2 -17433.87} C_VEL
LIN {X 0,Y 298.83,Z 541.321,A -85,B 0,C 180,E1 -17434.253,E2 -17434.253} C_VEL
LIN {X 0,Y 295.635,Z 550.352,A -85,B 0,C 180,E1 -17435.791,E2 -17435.791} C_VEL
LIN {X 0,Y 291.973,Z 559.623,A -85,B 0,C 180,E1 -17437.721,E2 -17437.721} C_VEL
LIN {X 0,Y 288.119,Z 568.545,A -85,B 0,C 180,E1 -17440.032,E2 -17440.032} C_VEL
LIN {X 0,Y 285.362,Z 574.673,A -85,B 0,C 180,E1 -17442.07,E2 -17442.07} C_VEL
LIN {X 0,Y 282.969,Z 579.722,A -85,B 0,C 180,E1 -17444.145,E2 -17444.145} C_VEL
LIN {X 0,Y 280.999,Z 583.704,A -85,B 0,C 180,E1 -17446.255,E2 -17446.255} C_VEL
LIN {X 0,Y 279.315,Z 586.735,A -85,B 0,C 180,E1 -17448.388,E2 -17448.388} C_VEL
LIN {X 0,Y 278.334,Z 588.419,A -85,B 0,C 180,E1 -17449.985,E2 -17449.985} C_VEL
LIN {X 0,Y 276.866,Z 590.166,A -85,B 0,C 180,E1 -17452.709,E2 -17452.709} C_VEL
LIN {X 0,Y 276.23,Z 590.517,A -85,B 0,C 180,E1 -17455.623,E2 -17455.623} C_VEL
LIN {X 0,Y 275.899,Z 590.099,A -85,B 0,C 180,E1 -17457.08,E2 -17457.08} C_VEL
LIN {X 0,Y 275.535,Z 588.089,A -85,B 0,C 180,E1 -17460,E2 -17460} C_VEL
LIN {X 0,Y 275.517,Z 585.51,A -85,B 0,C 180,E1 -17462.193,E2 -17462.193} C_VEL
LIN {X 0,Y 275.677,Z 581.96,A -85,B 0,C 180,E1 -17464.387,E2 -17464.387} C_VEL
LIN {X 0,Y 275.943,Z 576.564,A -85,B 0,C 180,E1 -17466.904,E2 -17466.904} C_VEL
LIN {X 0,Y 276.363,Z 570.382,A -85,B 0,C 180,E1 -17469.146,E2 -17469.146} C_VEL
LIN {X 0,Y 277.055,Z 562.903,A -85,B 0,C 180,E1 -17471.338,E2 -17471.338} C_VEL
LIN {X 0,Y 277.98,Z 553.765,A -85,B 0,C 180,E1 -17473.525,E2 -17473.525} C_VEL
LIN {X 0,Y 279.058,Z 543.444,A -85,B 0,C 180,E1 -17475.521,E2 -17475.521} C_VEL
LIN {X 0,Y 280.206,Z 533.256,A -85,B 0,C 180,E1 -17477.14,E2 -17477.14} C_VEL
LIN {X 0,Y 281.175,Z 522.404,A -85,B 0,C 180,E1 -17478.568,E2 -17478.568} C_VEL
LIN {X 0,Y 281.648,Z 515.735,A -85,B 0,C 180,E1 -17479.307,E2 -17479.307} C_VEL
LIN {X 0,Y 279.173,Z 502.51,A -85,B 0,C 180,E1 -17480.637,E2 -17480.637} C_VEL
LIN {X 0,Y 276.469,Z 488.131,A -85,B 0,C 180,E1 -17481.749,E2 -17481.749} C_VEL
LIN {X 0,Y 275.852,Z 484.564,A -85,B 0,C 180,E1 -17481.975,E2 -17481.975} C_VEL
LIN {X 0,Y 275.912,Z 482.768,A -85,B 0,C 180,E1 -17484.052,E2 -17484.052} C_VEL
LIN {X 0,Y 276.038,Z 482.103,A -85,B 0,C 180,E1 -17485.647,E2 -17485.647} C_VEL
LIN {X 0,Y 276.451,Z 482.047,A -85,B 0,C 180,E1 -17488.884,E2 -17488.884} C_VEL
LIN {X 0,Y 276.882,Z 481.991,A -85,B 0,C 180,E1 -17493.109,E2 -17493.109} C_VEL
LIN {X 0,Y 277.113,Z 481.965,A -85,B 0,C 180,E1 -17495.75,E2 -17495.75} C_VEL
LIN {X 0,Y 277.223,Z 481.95,A -85,B 0,C 180,E1 -17499.331,E2 -17499.331} C_VEL
LIN {X 0,Y 277.213,Z 481.951,A -85,B 0,C 180,E1 -17503.198,E2 -17503.198} C_VEL
LIN {X 0,Y 277.218,Z 481.951,A -85,B 0,C 180,E1 -17507.325,E2 -17507.325} C_VEL
LIN {X 0,Y 277.279,Z 481.944,A -85,B 0,C 180,E1 -17511.79,E2 -17511.79} C_VEL
LIN {X 0,Y 277.323,Z 481.941,A -85,B 0,C 180,E1 -17514.347,E2 -17514.347} C_VEL
LIN {X 0,Y 277.249,Z 481.949,A -85,B 0,C 180,E1 -17517.837,E2 -17517.837} C_VEL
LIN {X 0,Y 277.275,Z 481.943,A -85,B 0,C 180,E1 -17521.211,E2 -17521.211} C_VEL
LIN {X 0,Y 277.318,Z 481.94,A -85,B 0,C 180,E1 -17524.48,E2 -17524.48} C_VEL
LIN {X 0,Y 277.29,Z 481.942,A -85,B 0,C 180,E1 -17527.655,E2 -17527.655} C_VEL
LIN {X 0,Y 277.349,Z 481.935,A -85,B 0,C 180,E1 -17530.766,E2 -17530.766} C_VEL
LIN {X 0,Y 277.439,Z 481.923,A -85,B 0,C 180,E1 -17535.326,E2 -17535.326} C_VEL
LIN {X 0,Y 277.511,Z 481.917,A -85,B 0,C 180,E1 -17539.789,E2 -17539.789} C_VEL
LIN {X 0,Y 277.658,Z 481.896,A -85,B 0,C 180,E1 -17542.729,E2 -17542.729} C_VEL
LIN {X 0,Y 277.825,Z 481.876,A -85,B 0,C 180,E1 -17548.55,E2 -17548.55} C_VEL
LIN {X 0,Y 277.825,Z 481.876,A -85,B 0,C 180,E1 -17551.45,E2 -17551.45} C_VEL
LIN {X 0,Y 277.616,Z 481.901,A -85,B 0,C 180,E1 -17557.272,E2 -17557.272} C_VEL
LIN {X 0,Y 277.465,Z 481.922,A -85,B 0,C 180,E1 -17560.213,E2 -17560.213} C_VEL
LIN {X 0,Y 277.439,Z 481.923,A -85,B 0,C 180,E1 -17564.674,E2 -17564.674} C_VEL
LIN {X 0,Y 277.349,Z 481.935,A -85,B 0,C 180,E1 -17569.234,E2 -17569.234} C_VEL
LIN {X 0,Y 277.322,Z 481.94,A -85,B 0,C 180,E1 -17574.169,E2 -17574.169} C_VEL
LIN {X 0,Y 277.328,Z 481.939,A -85,B 0,C 180,E1 -17577.504,E2 -17577.504} C_VEL
LIN {X 0,Y 277.276,Z 481.943,A -85,B 0,C 180,E1 -17580.481,E2 -17580.481} C_VEL
LIN {X 0,Y 277.258,Z 481.95,A -85,B 0,C 180,E1 -17583.894,E2 -17583.894} C_VEL
LIN {X 0,Y 277.285,Z 481.945,A -85,B 0,C 180,E1 -17587.467,E2 -17587.467} C_VEL
LIN {X 0,Y 277.213,Z 481.952,A -85,B 0,C 180,E1 -17591.236,E2 -17591.236} C_VEL
LIN {X 0,Y 277.204,Z 481.954,A -85,B 0,C 180,E1 -17595.226,E2 -17595.226} C_VEL
LIN {X 0,Y 277.225,Z 481.952,A -85,B 0,C 180,E1 -17599.512,E2 -17599.512} C_VEL
LIN {X 0,Y 277.238,Z 481.949,A -85,B 0,C 180,E1 -17602.525,E2 -17602.525} C_VEL
LIN {X 0,Y 277.019,Z 481.976,A -85,B 0,C 180,E1 -17606.072,E2 -17606.072} C_VEL
LIN {X 0,Y 276.673,Z 482.023,A -85,B 0,C 180,E1 -17609.731,E2 -17609.731} C_VEL
LIN {X 0,Y 276.292,Z 482.066,A -85,B 0,C 180,E1 -17612.91,E2 -17612.91} C_VEL
LIN {X 0,Y 275.799,Z 482.305,A -85,B 0,C 180,E1 -17616.859,E2 -17616.859} C_VEL
LIN {X 0,Y 275.778,Z 483.653,A -85,B 0,C 180,E1 -17618.191,E2 -17618.191} C_VEL
LIN {X 0,Y 278.235,Z 497.48,A -85,B 0,C 180,E1 -17619.163,E2 -17619.163} C_VEL
LIN {X 0,Y 280.61,Z 510.279,A -85,B 0,C 180,E1 -17620.333,E2 -17620.333} C_VEL
LIN {X 0,Y 281.539,Z 515.349,A -85,B 0,C 180,E1 -17620.874,E2 -17620.874} C_VEL
LIN {X 0,Y 280.717,Z 526.141,A -85,B 0,C 180,E1 -17622.123,E2 -17622.123} C_VEL
LIN {X 0,Y 279.713,Z 536.529,A -85,B 0,C 180,E1 -17623.58,E2 -17623.58} C_VEL
LIN {X 0,Y 278.579,Z 547.104,A -85,B 0,C 180,E1 -17625.387,E2 -17625.387} C_VEL
LIN {X 0,Y 277.512,Z 557.482,A -85,B 0,C 180,E1 -17627.569,E2 -17627.569} C_VEL
LIN {X 0,Y 276.711,Z 565.87,A -85,B 0,C 180,E1 -17629.759,E2 -17629.759} C_VEL
LIN {X 0,Y 276.113,Z 572.709,A -85,B 0,C 180,E1 -17631.952,E2 -17631.952} C_VEL
LIN {X 0,Y 275.738,Z 578.236,A -85,B 0,C 180,E1 -17634.148,E2 -17634.148} C_VEL
LIN {X 0,Y 275.617,Z 582.576,A -85,B 0,C 180,E1 -17636.345,E2 -17636.345} C_VEL
LIN {X 0,Y 275.474,Z 585.845,A -85,B 0,C 180,E1 -17638.538,E2 -17638.538} C_VEL
LIN {X 0,Y 275.497,Z 587.497,A -85,B 0,C 180,E1 -17640,E2 -17640} C_VEL
LIN {X 0,Y 275.877,Z 589.541,A -85,B 0,C 180,E1 -17642.92,E2 -17642.92} C_VEL
LIN {X 0,Y 276.175,Z 589.996,A -85,B 0,C 180,E1 -17644.61,E2 -17644.61} C_VEL
LIN {X 0,Y 276.811,Z 589.667,A -85,B 0,C 180,E1 -17647.293,E2 -17647.293} C_VEL
LIN {X 0,Y 278.367,Z 587.801,A -85,B 0,C 180,E1 -17650.179,E2 -17650.179} C_VEL
LIN {X 0,Y 278.718,Z 587.033,A -85,B 0,C 180,E1 -17650.907,E2 -17650.907} C_VEL
LIN {X 0,Y 278.761,Z 585.828,A -85,B 0,C 180,E1 -17652.099,E2 -17652.099} C_VEL
LIN {X 0,Y 277.434,Z 583.705,A -85,B 0,C 180,E1 -17654.082,E2 -17654.082} C_VEL
LIN {X 0,Y 276.503,Z 580.995,A -85,B 0,C 180,E1 -17656.039,E2 -17656.039} C_VEL
LIN {X 0,Y 277.143,Z 578.833,A -85,B 0,C 180,E1 -17657.163,E2 -17657.163} C_VEL
LIN {X 0,Y 280.521,Z 572.196,A -85,B 0,C 180,E1 -17659.768,E2 -17659.768} C_VEL
LIN {X 0,Y 284.291,Z 564.269,A -85,B 0,C 180,E1 -17662.148,E2 -17662.148} C_VEL
LIN {X 0,Y 287.994,Z 555.948,A -85,B 0,C 180,E1 -17664.126,E2 -17664.126} C_VEL
LIN {X 0,Y 291.968,Z 545.905,A -85,B 0,C 180,E1 -17666.061,E2 -17666.061} C_VEL
LIN {X 0,Y 293.353,Z 542.295,A -85,B 0,C 180,E1 -17666.654,E2 -17666.654} C_VEL
LIN {X 0,Y 293.293,Z 538.017,A -85,B 0,C 180,E1 -17667.738,E2 -17667.738} C_VEL
LIN {X 0,Y 292.342,Z 531.763,A -85,B 0,C 180,E1 -17669.547,E2 -17669.547} C_VEL
LIN {X 0,Y 290.761,Z 525.56,A -85,B 0,C 180,E1 -17671.588,E2 -17671.588} C_VEL
LIN {X 0,Y 288.617,Z 519.342,A -85,B 0,C 180,E1 -17674.06,E2 -17674.06} C_VEL
LIN {X 0,Y 286.868,Z 515.65,A -85,B 0,C 180,E1 -17676.053,E2 -17676.053} C_VEL
LIN {X 0,Y 285.455,Z 512.795,A -85,B 0,C 180,E1 -17678.014,E2 -17678.014} C_VEL
LIN {X 0,Y 284.065,Z 511.279,A -85,B 0,C 180,E1 -17680.035,E2 -17680.035} C_VEL
LIN {X 0,Y 283.418,Z 510.006,A -85,B 0,C 180,E1 -17682.03,E2 -17682.03} C_VEL
LIN {X 0,Y 283.144,Z 509.602,A -85,B 0,C 180,E1 -17684.027,E2 -17684.027} C_VEL
LIN {X 0,Y 283.211,Z 510.342,A -85,B 0,C 180,E1 -17686.025,E2 -17686.025} C_VEL
LIN {X 0,Y 283.699,Z 512.06,A -85,B 0,C 180,E1 -17688.02,E2 -17688.02} C_VEL
LIN {X 0,Y 285.101,Z 516.076,A -85,B 0,C 180,E1 -17690.797,E2 -17690.797} C_VEL
LIN {X 0,Y 286.01,Z 518.581,A -85,B 0,C 180,E1 -17692.098,E2 -17692.098} C_VEL
LIN {X 0,Y 287.118,Z 524.073,A -85,B 0,C 180,E1 -17694.022,E2 -17694.022} C_VEL
LIN {X 0,Y 288.173,Z 530.51,A -85,B 0,C 180,E1 -17695.88,E2 -17695.88} C_VEL
LIN {X 0,Y 288.657,Z 539.141,A -85,B 0,C 180,E1 -17697.857,E2 -17697.857} C_VEL
LIN {X 0,Y 288.582,Z 550.13,A -85,B 0,C 180,E1 -17700.15,E2 -17700.15} C_VEL
LIN {X 0,Y 287.673,Z 561.066,A -85,B 0,C 180,E1 -17702.343,E2 -17702.343} C_VEL
LIN {X 0,Y 285.977,Z 570.083,A -85,B 0,C 180,E1 -17704.137,E2 -17704.137} C_VEL
LIN {X 0,Y 284.014,Z 576.818,A -85,B 0,C 180,E1 -17705.513,E2 -17705.513} C_VEL
LIN {X 0,Y 279.84,Z 587.303,A -85,B 0,C 180,E1 -17707.87,E2 -17707.87} C_VEL
LIN {X 0,Y 276.803,Z 594.716,A -85,B 0,C 180,E1 -17709.955,E2 -17709.955} C_VEL
LIN {X 0,Y 274.232,Z 600.962,A -85,B 0,C 180,E1 -17712.089,E2 -17712.089} C_VEL
LIN {X 0,Y 272.272,Z 606.109,A -85,B 0,C 180,E1 -17714.274,E2 -17714.274} C_VEL
LIN {X 0,Y 270.472,Z 610.297,A -85,B 0,C 180,E1 -17716.476,E2 -17716.476} C_VEL
LIN {X 0,Y 269.134,Z 614.385,A -85,B 0,C 180,E1 -17719.467,E2 -17719.467} C_VEL
LIN {X 0,Y 268.449,Z 616.967,A -85,B 0,C 180,E1 -17722.478,E2 -17722.478} C_VEL
LIN {X 0,Y 268.359,Z 617.936,A -85,B 0,C 180,E1 -17725.494,E2 -17725.494} C_VEL
LIN {X 0,Y 268.712,Z 617.348,A -85,B 0,C 180,E1 -17728.501,E2 -17728.501} C_VEL
LIN {X 0,Y 268.755,Z 617.144,A -85,B 0,C 180,E1 -17729.064,E2 -17729.064} C_VEL
LIN {X 0,Y 268.779,Z 617.949,A -85,B 0,C 180,E1 -17730,E2 -17730} C_VEL
LIN {X 0,Y 268.568,Z 618.848,A -85,B 0,C 180,E1 -17731.5,E2 -17731.5} C_VEL
LIN {X 0,Y 268.308,Z 619.422,A -85,B 0,C 180,E1 -17734.507,E2 -17734.507} C_VEL
LIN {X 0,Y 268.408,Z 618.444,A -85,B 0,C 180,E1 -17737.523,E2 -17737.523} C_VEL
LIN {X 0,Y 269.156,Z 615.883,A -85,B 0,C 180,E1 -17740.532,E2 -17740.532} C_VEL
LIN {X 0,Y 270.476,Z 611.811,A -85,B 0,C 180,E1 -17743.524,E2 -17743.524} C_VEL
LIN {X 0,Y 272.246,Z 607.67,A -85,B 0,C 180,E1 -17745.727,E2 -17745.727} C_VEL
LIN {X 0,Y 274.746,Z 601.203,A -85,B 0,C 180,E1 -17748.437,E2 -17748.437} C_VEL
LIN {X 0,Y 277.674,Z 594.148,A -85,B 0,C 180,E1 -17750.753,E2 -17750.753} C_VEL
LIN {X 0,Y 281.569,Z 584.955,A -85,B 0,C 180,E1 -17753.149,E2 -17753.149} C_VEL
LIN {X 0,Y 285.343,Z 575.526,A -85,B 0,C 180,E1 -17755.142,E2 -17755.142} C_VEL
LIN {X 0,Y 287.601,Z 566.816,A -85,B 0,C 180,E1 -17756.877,E2 -17756.877} C_VEL
LIN {X 0,Y 288.497,Z 557.997,A -85,B 0,C 180,E1 -17758.719,E2 -17758.719} C_VEL
LIN {X 0,Y 288.517,Z 548.681,A -85,B 0,C 180,E1 -17760.767,E2 -17760.767} C_VEL
LIN {X 0,Y 287.606,Z 538.889,A -85,B 0,C 180,E1 -17763.174,E2 -17763.174} C_VEL
LIN {X 0,Y 286.656,Z 532.309,A -85,B 0,C 180,E1 -17765.028,E2 -17765.028} C_VEL
LIN {X 0,Y 286.103,Z 528.728,A -85,B 0,C 180,E1 -17766.125,E2 -17766.125} C_VEL
LIN {X 0,Y 285.003,Z 523.575,A -85,B 0,C 180,E1 -17768.06,E2 -17768.06} C_VEL
LIN {X 0,Y 283.803,Z 520.362,A -85,B 0,C 180,E1 -17769.855,E2 -17769.855} C_VEL
LIN {X 0,Y 282.823,Z 515.837,A -85,B 0,C 180,E1 -17772.988,E2 -17772.988} C_VEL
LIN {X 0,Y 282.69,Z 514.746,A -85,B 0,C 180,E1 -17774.116,E2 -17774.116} C_VEL
LIN {X 0,Y 282.636,Z 513.879,A -85,B 0,C 180,E1 -17776.146,E2 -17776.146} C_VEL
LIN {X 0,Y 282.806,Z 514.419,A -85,B 0,C 180,E1 -17778.205,E2 -17778.205} C_VEL
LIN {X 0,Y 284.789,Z 516.25,A -85,B 0,C 180,E1 -17781.907,E2 -17781.907} C_VEL
LIN {X 0,Y 286.392,Z 519.001,A -85,B 0,C 180,E1 -17784.078,E2 -17784.078} C_VEL
LIN {X 0,Y 288.09,Z 522.405,A -85,B 0,C 180,E1 -17786.041,E2 -17786.041} C_VEL
LIN {X 0,Y 289.909,Z 526.863,A -85,B 0,C 180,E1 -17788.046,E2 -17788.046} C_VEL
LIN {X 0,Y 291.698,Z 532.6,A -85,B 0,C 180,E1 -17790.154,E2 -17790.154} C_VEL
LIN {X 0,Y 292.968,Z 538.65,A -85,B 0,C 180,E1 -17792.081,E2 -17792.081} C_VEL
LIN {X 0,Y 293.473,Z 543.092,A -85,B 0,C 180,E1 -17793.342,E2 -17793.342} C_VEL
LIN {X 0,Y 289.584,Z 553.399,A -85,B 0,C 180,E1 -17795.251,E2 -17795.251} C_VEL
LIN {X 0,Y 285.764,Z 562.236,A -85,B 0,C 180,E1 -17797.21,E2 -17797.21} C_VEL
LIN {X 0,Y 281.705,Z 570.635,A -85,B 0,C 180,E1 -17799.557,E2 -17799.557} C_VEL
LIN {X 0,Y 278.826,Z 576.485,A -85,B 0,C 180,E1 -17801.635,E2 -17801.635} C_VEL
LIN {X 0,Y 276.299,Z 581.216,A -85,B 0,C 180,E1 -17803.752,E2 -17803.752} C_VEL
LIN {X 0,Y 273.495,Z 586.06,A -85,B 0,C 180,E1 -17806.628,E2 -17806.628} C_VEL
LIN {X 0,Y 271.515,Z 589.193,A -85,B 0,C 180,E1 -17809.561,E2 -17809.561} C_VEL
LIN {X 0,Y 269.87,Z 590.868,A -85,B 0,C 180,E1 -17812.519,E2 -17812.519} C_VEL
LIN {X 0,Y 269.48,Z 591.107,A -85,B 0,C 180,E1 -17814.012,E2 -17814.012} C_VEL
LIN {X 0,Y 269.163,Z 590.951,A -85,B 0,C 180,E1 -17815.508,E2 -17815.508} C_VEL
LIN {X 0,Y 268.581,Z 589.527,A -85,B 0,C 180,E1 -17818.501,E2 -17818.501} C_VEL
LIN {X 0,Y 268.448,Z 588.226,A -85,B 0,C 180,E1 -17820,E2 -17820} C_VEL
LIN {X 0,Y 268.442,Z 585.476,A -85,B 0,C 180,E1 -17822.251,E2 -17822.251} C_VEL
LIN {X 0,Y 268.578,Z 581.74,A -85,B 0,C 180,E1 -17824.503,E2 -17824.503} C_VEL
LIN {X 0,Y 268.862,Z 576.411,A -85,B 0,C 180,E1 -17826.964,E2 -17826.964} C_VEL
LIN {X 0,Y 269.34,Z 569.746,A -85,B 0,C 180,E1 -17829.386,E2 -17829.386} C_VEL
LIN {X 0,Y 270.065,Z 562.056,A -85,B 0,C 180,E1 -17831.636,E2 -17831.636} C_VEL
LIN {X 0,Y 271.014,Z 552.567,A -85,B 0,C 180,E1 -17833.88,E2 -17833.88} C_VEL
LIN {X 0,Y 272.111,Z 541.922,A -85,B 0,C 180,E1 -17835.928,E2 -17835.928} C_VEL
LIN {X 0,Y 273.212,Z 532.624,A -85,B 0,C 180,E1 -17837.4,E2 -17837.4} C_VEL
LIN {X 0,Y 274.251,Z 521.36,A -85,B 0,C 180,E1 -17838.876,E2 -17838.876} C_VEL
LIN {X 0,Y 274.574,Z 516.433,A -85,B 0,C 180,E1 -17839.436,E2 -17839.436} C_VEL
LIN {X 0,Y 272.116,Z 503.255,A -85,B 0,C 180,E1 -17840.807,E2 -17840.807} C_VEL
LIN {X 0,Y 269.521,Z 489.265,A -85,B 0,C 180,E1 -17841.935,E2 -17841.935} C_VEL
LIN {X 0,Y 268.807,Z 484.925,A -85,B 0,C 180,E1 -17842.242,E2 -17842.242} C_VEL
LIN {X 0,Y 268.869,Z 482.997,A -85,B 0,C 180,E1 -17844.723,E2 -17844.723} C_VEL
LIN {X 0,Y 269.278,Z 482.946,A -85,B 0,C 180,E1 -17848.021,E2 -17848.021} C_VEL
LIN {X 0,Y 269.624,Z 482.896,A -85,B 0,C 180,E1 -17851.421,E2 -17851.421} C_VEL
LIN {X 0,Y 269.973,Z 482.854,A -85,B 0,C 180,E1 -17854.94,E2 -17854.94} C_VEL
LIN {X 0,Y 270.17,Z 482.83,A -85,B 0,C 180,E1 -17858.703,E2 -17858.703} C_VEL
LIN {X 0,Y 270.175,Z 482.83,A -85,B 0,C 180,E1 -17862.558,E2 -17862.558} C_VEL
LIN {X 0,Y 270.168,Z 482.83,A -85,B 0,C 180,E1 -17866.751,E2 -17866.751} C_VEL
LIN {X 0,Y 270.226,Z 482.82,A -85,B 0,C 180,E1 -17871.283,E2 -17871.283} C_VEL
LIN {X 0,Y 270.227,Z 482.822,A -85,B 0,C 180,E1 -17875.098,E2 -17875.098} C_VEL
LIN {X 0,Y 270.204,Z 482.823,A -85,B 0,C 180,E1 -17879.131,E2 -17879.131} C_VEL
LIN {X 0,Y 270.268,Z 482.821,A -85,B 0,C 180,E1 -17882.146,E2 -17882.146} C_VEL
LIN {X 0,Y 270.281,Z 482.815,A -85,B 0,C 180,E1 -17885.519,E2 -17885.519} C_VEL
LIN {X 0,Y 270.306,Z 482.816,A -85,B 0,C 180,E1 -17890.245,E2 -17890.245} C_VEL
LIN {X 0,Y 270.408,Z 482.799,A -85,B 0,C 180,E1 -17894.936,E2 -17894.936} C_VEL
LIN {X 0,Y 270.446,Z 482.795,A -85,B 0,C 180,E1 -17899.519,E2 -17899.519} C_VEL
LIN {X 0,Y 270.617,Z 482.774,A -85,B 0,C 180,E1 -17902.539,E2 -17902.539} C_VEL
LIN {X 0,Y 270.791,Z 482.753,A -85,B 0,C 180,E1 -17908.513,E2 -17908.513} C_VEL
LIN {X 0,Y 270.791,Z 482.753,A -85,B 0,C 180,E1 -17911.487,E2 -17911.487} C_VEL
LIN {X 0,Y 270.575,Z 482.779,A -85,B 0,C 180,E1 -17917.462,E2 -17917.462} C_VEL
LIN {X 0,Y 270.417,Z 482.799,A -85,B 0,C 180,E1 -17920.482,E2 -17920.482} C_VEL
LIN {X 0,Y 270.408,Z 482.799,A -85,B 0,C 180,E1 -17925.064,E2 -17925.064} C_VEL
LIN {X 0,Y 270.305,Z 482.816,A -85,B 0,C 180,E1 -17929.755,E2 -17929.755} C_VEL
LIN {X 0,Y 270.277,Z 482.816,A -85,B 0,C 180,E1 -17934.585,E2 -17934.585} C_VEL
LIN {X 0,Y 270.274,Z 482.82,A -85,B 0,C 180,E1 -17937.909,E2 -17937.909} C_VEL
LIN {X 0,Y 270.188,Z 482.826,A -85,B 0,C 180,E1 -17941.348,E2 -17941.348} C_VEL
LIN {X 0,Y 270.227,Z 482.822,A -85,B 0,C 180,E1 -17944.902,E2 -17944.902} C_VEL
LIN {X 0,Y 270.226,Z 482.82,A -85,B 0,C 180,E1 -17948.717,E2 -17948.717} C_VEL
LIN {X 0,Y 270.169,Z 482.83,A -85,B 0,C 180,E1 -17953.249,E2 -17953.249} C_VEL
LIN {X 0,Y 270.175,Z 482.83,A -85,B 0,C 180,E1 -17957.442,E2 -17957.442} C_VEL
LIN {X 0,Y 270.21,Z 482.826,A -85,B 0,C 180,E1 -17961.374,E2 -17961.374} C_VEL
LIN {X 0,Y 270.038,Z 482.846,A -85,B 0,C 180,E1 -17965.07,E2 -17965.07} C_VEL
LIN {X 0,Y 269.963,Z 482.853,A -85,B 0,C 180,E1 -17966.859,E2 -17966.859} C_VEL
LIN {X 0,Y 269.537,Z 482.908,A -85,B 0,C 180,E1 -17970.302,E2 -17970.302} C_VEL
LIN {X 0,Y 269.124,Z 482.963,A -85,B 0,C 180,E1 -17973.644,E2 -17973.644} C_VEL
LIN {X 0,Y 268.726,Z 483.173,A -85,B 0,C 180,E1 -17977.106,E2 -17977.106} C_VEL
LIN {X 0,Y 268.719,Z 483.996,A -85,B 0,C 180,E1 -17977.941,E2 -17977.941} C_VEL
LIN {X 0,Y 271.364,Z 499.19,A -85,B 0,C 180,E1 -17979.063,E2 -17979.063} C_VEL
LIN {X 0,Y 273.799,Z 512.455,A -85,B 0,C 180,E1 -17980.351,E2 -17980.351} C_VEL
LIN {X 0,Y 274.461,Z 516.027,A -85,B 0,C 180,E1 -17980.75,E2 -17980.75} C_VEL
LIN {X 0,Y 273.737,Z 525.47,A -85,B 0,C 180,E1 -17981.862,E2 -17981.862} C_VEL
LIN {X 0,Y 272.728,Z 535.915,A -85,B 0,C 180,E1 -17983.34,E2 -17983.34} C_VEL
LIN {X 0,Y 271.677,Z 545.707,A -85,B 0,C 180,E1 -17985.007,E2 -17985.007} C_VEL
LIN {X 0,Y 270.652,Z 554.796,A -85,B 0,C 180,E1 -17986.867,E2 -17986.867} C_VEL
LIN {X 0,Y 269.788,Z 563.776,A -85,B 0,C 180,E1 -17989.113,E2 -17989.113} C_VEL
LIN {X 0,Y 269.15,Z 571.095,A -85,B 0,C 180,E1 -17991.364,E2 -17991.364} C_VEL
LIN {X 0,Y 268.714,Z 577.068,A -85,B 0,C 180,E1 -17993.649,E2 -17993.649} C_VEL
LIN {X 0,Y 268.534,Z 582.354,A -85,B 0,C 180,E1 -17996.248,E2 -17996.248} C_VEL
LIN {X 0,Y 268.394,Z 585.812,A -85,B 0,C 180,E1 -17998.499,E2 -17998.499} C_VEL
LIN {X 0,Y 268.412,Z 587.586,A -85,B 0,C 180,E1 -18000,E2 -18000} C_VEL
LIN {X 0,Y 268.537,Z 588.943,A -85,B 0,C 180,E1 -18001.499,E2 -18001.499} C_VEL
LIN {X 0,Y 268.799,Z 589.856,A -85,B 0,C 180,E1 -18002.997,E2 -18002.997} C_VEL
LIN {X 0,Y 269.079,Z 590.397,A -85,B 0,C 180,E1 -18004.494,E2 -18004.494} C_VEL
LIN {X 0,Y 269.819,Z 590.352,A -85,B 0,C 180,E1 -18007.483,E2 -18007.483} C_VEL
LIN {X 0,Y 271.452,Z 588.687,A -85,B 0,C 180,E1 -18010.441,E2 -18010.441} C_VEL
LIN {X 0,Y 272.233,Z 587.344,A -85,B 0,C 180,E1 -18011.919,E2 -18011.919} C_VEL
LIN {X 0,Y 274.061,Z 584.494,A -85,B 0,C 180,E1 -18014.1,E2 -18014.1} C_VEL
LIN {X 0,Y 276.094,Z 580.736,A -85,B 0,C 180,E1 -18016.26,E2 -18016.26} C_VEL
LIN {X 0,Y 277.143,Z 578.833,A -85,B 0,C 180,E1 -18017.163,E2 -18017.163} C_VEL
LIN {X 0,Y 277.883,Z 576.513,A -85,B 0,C 180,E1 -18018.276,E2 -18018.276} C_VEL
LIN {X 0,Y 277.599,Z 572.803,A -85,B 0,C 180,E1 -18020.176,E2 -18020.176} C_VEL
LIN {X 0,Y 277.57,Z 568.575,A -85,B 0,C 180,E1 -18022.017,E2 -18022.017} C_VEL
LIN {X 0,Y 278.662,Z 565.444,A -85,B 0,C 180,E1 -18023.016,E2 -18023.016} C_VEL
LIN {X 0,Y 283.238,Z 555.879,A -85,B 0,C 180,E1 -18025.342,E2 -18025.342} C_VEL
LIN {X 0,Y 287.49,Z 545.979,A -85,B 0,C 180,E1 -18027.242,E2 -18027.242} C_VEL
LIN {X 0,Y 288.007,Z 544.089,A -85,B 0,C 180,E1 -18027.622,E2 -18027.622} C_VEL
LIN {X 0,Y 287.707,Z 538.643,A -85,B 0,C 180,E1 -18029.245,E2 -18029.245} C_VEL
LIN {X 0,Y 286.686,Z 532.456,A -85,B 0,C 180,E1 -18031.316,E2 -18031.316} C_VEL
LIN {X 0,Y 285.07,Z 526.286,A -85,B 0,C 180,E1 -18033.784,E2 -18033.784} C_VEL
LIN {X 0,Y 283.483,Z 522.057,A -85,B 0,C 180,E1 -18036.044,E2 -18036.044} C_VEL
LIN {X 0,Y 281.906,Z 518.775,A -85,B 0,C 180,E1 -18038.554,E2 -18038.554} C_VEL
LIN {X 0,Y 280.621,Z 516.938,A -85,B 0,C 180,E1 -18041.294,E2 -18041.294} C_VEL
LIN {X 0,Y 280.345,Z 516.204,A -85,B 0,C 180,E1 -18043.364,E2 -18043.364} C_VEL
LIN {X 0,Y 280.34,Z 516.633,A -85,B 0,C 180,E1 -18045.416,E2 -18045.416} C_VEL
LIN {X 0,Y 280.678,Z 518.127,A -85,B 0,C 180,E1 -18047.463,E2 -18047.463} C_VEL
LIN {X 0,Y 281.29,Z 520.727,A -85,B 0,C 180,E1 -18049.488,E2 -18049.488} C_VEL
LIN {X 0,Y 282.429,Z 524.023,A -85,B 0,C 180,E1 -18051.53,E2 -18051.53} C_VEL
LIN {X 0,Y 283.316,Z 530.35,A -85,B 0,C 180,E1 -18053.808,E2 -18053.808} C_VEL
LIN {X 0,Y 283.792,Z 535.238,A -85,B 0,C 180,E1 -18055.278,E2 -18055.278} C_VEL
LIN {X 0,Y 283.79,Z 543.826,A -85,B 0,C 180,E1 -18057.352,E2 -18057.352} C_VEL
LIN {X 0,Y 283.235,Z 553.692,A -85,B 0,C 180,E1 -18059.542,E2 -18059.542} C_VEL
LIN {X 0,Y 281.917,Z 563.867,A -85,B 0,C 180,E1 -18061.728,E2 -18061.728} C_VEL
LIN {X 0,Y 280.437,Z 570.748,A -85,B 0,C 180,E1 -18063.186,E2 -18063.186} C_VEL
LIN {X 0,Y 277.745,Z 578.792,A -85,B 0,C 180,E1 -18064.923,E2 -18064.923} C_VEL
LIN {X 0,Y 273.987,Z 587.398,A -85,B 0,C 180,E1 -18066.972,E2 -18066.972} C_VEL
LIN {X 0,Y 270.337,Z 595.529,A -85,B 0,C 180,E1 -18069.374,E2 -18069.374} C_VEL
LIN {X 0,Y 267.539,Z 601.666,A -85,B 0,C 180,E1 -18071.625,E2 -18071.625} C_VEL
LIN {X 0,Y 265.472,Z 606.556,A -85,B 0,C 180,E1 -18073.861,E2 -18073.861} C_VEL
LIN {X 0,Y 263.568,Z 610.496,A -85,B 0,C 180,E1 -18076.114,E2 -18076.114} C_VEL
LIN {X 0,Y 262.115,Z 614.367,A -85,B 0,C 180,E1 -18079.182,E2 -18079.182} C_VEL
LIN {X 0,Y 261.373,Z 616.657,A -85,B 0,C 180,E1 -18082.274,E2 -18082.274} C_VEL
LIN {X 0,Y 261.284,Z 617.44,A -85,B 0,C 180,E1 -18085.372,E2 -18085.372} C_VEL
LIN {X 0,Y 261.345,Z 617.242,A -85,B 0,C 180,E1 -18086.917,E2 -18086.917} C_VEL
LIN {X 0,Y 261.719,Z 616.36,A -85,B 0,C 180,E1 -18089.135,E2 -18089.135} C_VEL
LIN {X 0,Y 261.502,Z 618.134,A -85,B 0,C 180,E1 -18091.54,E2 -18091.54} C_VEL
LIN {X 0,Y 261.276,Z 618.729,A -85,B 0,C 180,E1 -18093.084,E2 -18093.084} C_VEL
LIN {X 0,Y 261.212,Z 618.859,A -85,B 0,C 180,E1 -18095.439,E2 -18095.439} C_VEL
LIN {X 0,Y 261.342,Z 618.116,A -85,B 0,C 180,E1 -18097.727,E2 -18097.727} C_VEL
LIN {X 0,Y 262.135,Z 615.837,A -85,B 0,C 180,E1 -18100.817,E2 -18100.817} C_VEL
LIN {X 0,Y 263.57,Z 611.996,A -85,B 0,C 180,E1 -18103.886,E2 -18103.886} C_VEL
LIN {X 0,Y 266.07,Z 606.603,A -85,B 0,C 180,E1 -18106.891,E2 -18106.891} C_VEL
LIN {X 0,Y 268.668,Z 600.595,A -85,B 0,C 180,E1 -18109.443,E2 -18109.443} C_VEL
LIN {X 0,Y 272.778,Z 591.729,A -85,B 0,C 180,E1 -18112.335,E2 -18112.335} C_VEL
LIN {X 0,Y 276.479,Z 583.696,A -85,B 0,C 180,E1 -18114.398,E2 -18114.398} C_VEL
LIN {X 0,Y 279.736,Z 575.974,A -85,B 0,C 180,E1 -18116.083,E2 -18116.083} C_VEL
LIN {X 0,Y 281.693,Z 569.32,A -85,B 0,C 180,E1 -18117.488,E2 -18117.488} C_VEL
LIN {X 0,Y 282.876,Z 561.25,A -85,B 0,C 180,E1 -18119.293,E2 -18119.293} C_VEL
LIN {X 0,Y 283.3,Z 552.298,A -85,B 0,C 180,E1 -18121.397,E2 -18121.397} C_VEL
LIN {X 0,Y 282.887,Z 543.171,A -85,B 0,C 180,E1 -18123.801,E2 -18123.801} C_VEL
LIN {X 0,Y 282.147,Z 535.371,A -85,B 0,C 180,E1 -18126.192,E2 -18126.192} C_VEL
LIN {X 0,Y 281.514,Z 531.503,A -85,B 0,C 180,E1 -18127.618,E2 -18127.618} C_VEL
LIN {X 0,Y 280.971,Z 527.943,A -85,B 0,C 180,E1 -18129.158,E2 -18129.158} C_VEL
LIN {X 0,Y 279.758,Z 522.779,A -85,B 0,C 180,E1 -18132.71,E2 -18132.71} C_VEL
LIN {X 0,Y 279.638,Z 520.901,A -85,B 0,C 180,E1 -18134.726,E2 -18134.726} C_VEL
LIN {X 0,Y 279.607,Z 520.53,A -85,B 0,C 180,E1 -18137.262,E2 -18137.262} C_VEL
LIN {X 0,Y 280.807,Z 522.017,A -85,B 0,C 180,E1 -18140.884,E2 -18140.884} C_VEL
LIN {X 0,Y 282.3,Z 524.277,A -85,B 0,C 180,E1 -18143.31,E2 -18143.31} C_VEL
LIN {X 0,Y 283.694,Z 527.195,A -85,B 0,C 180,E1 -18145.265,E2 -18145.265} C_VEL
LIN {X 0,Y 285.474,Z 532.175,A -85,B 0,C 180,E1 -18147.728,E2 -18147.728} C_VEL
LIN {X 0,Y 286.738,Z 536.853,A -85,B 0,C 180,E1 -18149.584,E2 -18149.584} C_VEL
LIN {X 0,Y 287.783,Z 543.793,A -85,B 0,C 180,E1 -18151.931,E2 -18151.931} C_VEL
LIN {X 0,Y 287.657,Z 547.04,A -85,B 0,C 180,E1 -18152.848,E2 -18152.848} C_VEL
LIN {X 0,Y 283.55,Z 556.545,A -85,B 0,C 180,E1 -18154.688,E2 -18154.688} C_VEL
LIN {X 0,Y 278.934,Z 566.042,A -85,B 0,C 180,E1 -18157.012,E2 -18157.012} C_VEL
LIN {X 0,Y 275.354,Z 572.796,A -85,B 0,C 180,E1 -18159.064,E2 -18159.064} C_VEL
LIN {X 0,Y 272.324,Z 578.267,A -85,B 0,C 180,E1 -18161.18,E2 -18161.18} C_VEL
LIN {X 0,Y 269.679,Z 582.764,A -85,B 0,C 180,E1 -18163.342,E2 -18163.342} C_VEL
LIN {X 0,Y 267.469,Z 586.255,A -85,B 0,C 180,E1 -18165.545,E2 -18165.545} C_VEL
LIN {X 0,Y 265.612,Z 588.858,A -85,B 0,C 180,E1 -18167.78,E2 -18167.78} C_VEL
LIN {X 0,Y 264.49,Z 590.272,A -85,B 0,C 180,E1 -18169.472,E2 -18169.472} C_VEL
LIN {X 0,Y 262.879,Z 591.519,A -85,B 0,C 180,E1 -18172.318,E2 -18172.318} C_VEL
LIN {X 0,Y 262.099,Z 591.368,A -85,B 0,C 180,E1 -18175.386,E2 -18175.386} C_VEL
LIN {X 0,Y 261.747,Z 590.745,A -85,B 0,C 180,E1 -18176.922,E2 -18176.922} C_VEL
LIN {X 0,Y 261.498,Z 589.71,A -85,B 0,C 180,E1 -18178.46,E2 -18178.46} C_VEL
LIN {X 0,Y 261.342,Z 586.438,A -85,B 0,C 180,E1 -18181.541,E2 -18181.541} C_VEL
LIN {X 0,Y 261.457,Z 582.864,A -85,B 0,C 180,E1 -18183.854,E2 -18183.854} C_VEL
LIN {X 0,Y 261.678,Z 577.657,A -85,B 0,C 180,E1 -18186.42,E2 -18186.42} C_VEL
LIN {X 0,Y 262.12,Z 571.3,A -85,B 0,C 180,E1 -18188.869,E2 -18188.869} C_VEL
LIN {X 0,Y 262.769,Z 563.857,A -85,B 0,C 180,E1 -18191.181,E2 -18191.181} C_VEL
LIN {X 0,Y 263.693,Z 554.787,A -85,B 0,C 180,E1 -18193.486,E2 -18193.486} C_VEL
LIN {X 0,Y 264.87,Z 544.595,A -85,B 0,C 180,E1 -18195.585,E2 -18195.585} C_VEL
LIN {X 0,Y 266.126,Z 533.568,A -85,B 0,C 180,E1 -18197.428,E2 -18197.428} C_VEL
LIN {X 0,Y 267.153,Z 522.019,A -85,B 0,C 180,E1 -18198.999,E2 -18198.999} C_VEL
LIN {X 0,Y 267.512,Z 517.138,A -85,B 0,C 180,E1 -18199.571,E2 -18199.571} C_VEL
LIN {X 0,Y 265.07,Z 504.061,A -85,B 0,C 180,E1 -18200.979,E2 -18200.979} C_VEL
LIN {X 0,Y 262.569,Z 490.318,A -85,B 0,C 180,E1 -18202.137,E2 -18202.137} C_VEL
LIN {X 0,Y 261.729,Z 485.311,A -85,B 0,C 180,E1 -18202.498,E2 -18202.498} C_VEL
LIN {X 0,Y 261.798,Z 483.88,A -85,B 0,C 180,E1 -18204.317,E2 -18204.317} C_VEL
LIN {X 0,Y 262.216,Z 483.826,A -85,B 0,C 180,E1 -18207.812,E2 -18207.812} C_VEL
LIN {X 0,Y 262.557,Z 483.777,A -85,B 0,C 180,E1 -18211.067,E2 -18211.067} C_VEL
LIN {X 0,Y 262.86,Z 483.741,A -85,B 0,C 180,E1 -18214.158,E2 -18214.158} C_VEL
LIN {X 0,Y 263.061,Z 483.716,A -85,B 0,C 180,E1 -18217.914,E2 -18217.914} C_VEL
LIN {X 0,Y 263.127,Z 483.706,A -85,B 0,C 180,E1 -18221.894,E2 -18221.894} C_VEL
LIN {X 0,Y 263.127,Z 483.71,A -85,B 0,C 180,E1 -18226.151,E2 -18226.151} C_VEL
LIN {X 0,Y 263.119,Z 483.71,A -85,B 0,C 180,E1 -18230.13,E2 -18230.13} C_VEL
LIN {X 0,Y 263.194,Z 483.701,A -85,B 0,C 180,E1 -18234.023,E2 -18234.023} C_VEL
LIN {X 0,Y 263.138,Z 483.706,A -85,B 0,C 180,E1 -18237.712,E2 -18237.712} C_VEL
LIN {X 0,Y 263.203,Z 483.698,A -85,B 0,C 180,E1 -18241.784,E2 -18241.784} C_VEL
LIN {X 0,Y 263.23,Z 483.693,A -85,B 0,C 180,E1 -18245.2,E2 -18245.2} C_VEL
LIN {X 0,Y 263.268,Z 483.689,A -85,B 0,C 180,E1 -18249.694,E2 -18249.694} C_VEL
LIN {X 0,Y 263.355,Z 483.678,A -85,B 0,C 180,E1 -18254.522,E2 -18254.522} C_VEL
LIN {X 0,Y 263.379,Z 483.674,A -85,B 0,C 180,E1 -18259.235,E2 -18259.235} C_VEL
LIN {X 0,Y 263.578,Z 483.652,A -85,B 0,C 180,E1 -18262.339,E2 -18262.339} C_VEL
LIN {X 0,Y 263.756,Z 483.629,A -85,B 0,C 180,E1 -18268.473,E2 -18268.473} C_VEL
LIN {X 0,Y 263.755,Z 483.629,A -85,B 0,C 180,E1 -18271.527,E2 -18271.527} C_VEL
LIN {X 0,Y 263.537,Z 483.657,A -85,B 0,C 180,E1 -18277.663,E2 -18277.663} C_VEL
LIN {X 0,Y 263.359,Z 483.677,A -85,B 0,C 180,E1 -18280.766,E2 -18280.766} C_VEL
LIN {X 0,Y 263.355,Z 483.678,A -85,B 0,C 180,E1 -18285.478,E2 -18285.478} C_VEL
LIN {X 0,Y 263.267,Z 483.689,A -85,B 0,C 180,E1 -18290.306,E2 -18290.306} C_VEL
LIN {X 0,Y 263.212,Z 483.696,A -85,B 0,C 180,E1 -18295.291,E2 -18295.291} C_VEL
LIN {X 0,Y 263.179,Z 483.699,A -85,B 0,C 180,E1 -18298.73,E2 -18298.73} C_VEL
LIN {X 0,Y 263.137,Z 483.706,A -85,B 0,C 180,E1 -18302.288,E2 -18302.288} C_VEL
LIN {X 0,Y 263.194,Z 483.701,A -85,B 0,C 180,E1 -18305.977,E2 -18305.977} C_VEL
LIN {X 0,Y 263.119,Z 483.71,A -85,B 0,C 180,E1 -18309.87,E2 -18309.87} C_VEL
LIN {X 0,Y 263.126,Z 483.709,A -85,B 0,C 180,E1 -18313.984,E2 -18313.984} C_VEL
LIN {X 0,Y 263.127,Z 483.705,A -85,B 0,C 180,E1 -18318.406,E2 -18318.406} C_VEL
LIN {X 0,Y 263.121,Z 483.709,A -85,B 0,C 180,E1 -18322.096,E2 -18322.096} C_VEL
LIN {X 0,Y 262.958,Z 483.728,A -85,B 0,C 180,E1 -18325.948,E2 -18325.948} C_VEL
LIN {X 0,Y 262.619,Z 483.771,A -85,B 0,C 180,E1 -18329.438,E2 -18329.438} C_VEL
LIN {X 0,Y 262.194,Z 483.823,A -85,B 0,C 180,E1 -18332.891,E2 -18332.891} C_VEL
LIN {X 0,Y 261.654,Z 483.967,A -85,B 0,C 180,E1 -18337.287,E2 -18337.287} C_VEL
LIN {X 0,Y 261.66,Z 484.513,A -85,B 0,C 180,E1 -18337.704,E2 -18337.704} C_VEL
LIN {X 0,Y 264.239,Z 499.483,A -85,B 0,C 180,E1 -18338.838,E2 -18338.838} C_VEL
LIN {X 0,Y 266.677,Z 512.75,A -85,B 0,C 180,E1 -18340.165,E2 -18340.165} C_VEL
LIN {X 0,Y 267.38,Z 516.703,A -85,B 0,C 180,E1 -18340.619,E2 -18340.619} C_VEL
LIN {X 0,Y 266.518,Z 527.256,A -85,B 0,C 180,E1 -18341.917,E2 -18341.917} C_VEL
LIN {X 0,Y 265.57,Z 536.48,A -85,B 0,C 180,E1 -18343.274,E2 -18343.274} C_VEL
LIN {X 0,Y 264.565,Z 546.244,A -85,B 0,C 180,E1 -18344.989,E2 -18344.989} C_VEL
LIN {X 0,Y 263.537,Z 555.253,A -85,B 0,C 180,E1 -18346.898,E2 -18346.898} C_VEL
LIN {X 0,Y 262.669,Z 564.174,A -85,B 0,C 180,E1 -18349.205,E2 -18349.205} C_VEL
LIN {X 0,Y 262.017,Z 571.488,A -85,B 0,C 180,E1 -18351.516,E2 -18351.516} C_VEL
LIN {X 0,Y 261.592,Z 577.414,A -85,B 0,C 180,E1 -18353.83,E2 -18353.83} C_VEL
LIN {X 0,Y 261.451,Z 582.133,A -85,B 0,C 180,E1 -18356.146,E2 -18356.146} C_VEL
LIN {X 0,Y 261.317,Z 585.767,A -85,B 0,C 180,E1 -18358.458,E2 -18358.458} C_VEL
LIN {X 0,Y 261.457,Z 589.077,A -85,B 0,C 180,E1 -18361.54,E2 -18361.54} C_VEL
LIN {X 0,Y 261.724,Z 590.153,A -85,B 0,C 180,E1 -18363.078,E2 -18363.078} C_VEL
LIN {X 0,Y 262.017,Z 590.801,A -85,B 0,C 180,E1 -18364.615,E2 -18364.615} C_VEL
LIN {X 0,Y 262.83,Z 590.971,A -85,B 0,C 180,E1 -18367.683,E2 -18367.683} C_VEL
LIN {X 0,Y 264.205,Z 589.949,A -85,B 0,C 180,E1 -18370.19,E2 -18370.19} C_VEL
LIN {X 0,Y 265.361,Z 588.361,A -85,B 0,C 180,E1 -18372.232,E2 -18372.232} C_VEL
LIN {X 0,Y 268.018,Z 584.702,A -85,B 0,C 180,E1 -18375.202,E2 -18375.202} C_VEL
LIN {X 0,Y 270.643,Z 580.32,A -85,B 0,C 180,E1 -18377.659,E2 -18377.659} C_VEL
LIN {X 0,Y 274.11,Z 574.176,A -85,B 0,C 180,E1 -18380.251,E2 -18380.251} C_VEL
LIN {X 0,Y 277.451,Z 567.87,A -85,B 0,C 180,E1 -18382.331,E2 -18382.331} C_VEL
LIN {X 0,Y 278.662,Z 565.444,A -85,B 0,C 180,E1 -18383.016,E2 -18383.016} C_VEL
LIN {X 0,Y 280.742,Z 559.877,A -85,B 0,C 180,E1 -18384.612,E2 -18384.612} C_VEL
LIN {X 0,Y 281.411,Z 556.583,A -85,B 0,C 180,E1 -18385.6,E2 -18385.6} C_VEL
LIN {X 0,Y 282.503,Z 547.615,A -85,B 0,C 180,E1 -18388.248,E2 -18388.248} C_VEL
LIN {X 0,Y 282.56,Z 542.586,A -85,B 0,C 180,E1 -18389.831,E2 -18389.831} C_VEL
LIN {X 0,Y 281.83,Z 536.591,A -85,B 0,C 180,E1 -18392.02,E2 -18392.02} C_VEL
LIN {X 0,Y 280.755,Z 531.397,A -85,B 0,C 180,E1 -18394.302,E2 -18394.302} C_VEL
LIN {X 0,Y 279.574,Z 527.687,A -85,B 0,C 180,E1 -18396.445,E2 -18396.445} C_VEL
LIN {X 0,Y 278.508,Z 525.096,A -85,B 0,C 180,E1 -18398.531,E2 -18398.531} C_VEL
LIN {X 0,Y 277.448,Z 523.345,A -85,B 0,C 180,E1 -18401.193,E2 -18401.193} C_VEL
LIN {X 0,Y 277.23,Z 522.604,A -85,B 0,C 180,E1 -18403.194,E2 -18403.194} C_VEL
LIN {X 0,Y 277.228,Z 522.962,A -85,B 0,C 180,E1 -18405.221,E2 -18405.221} C_VEL
LIN {X 0,Y 277.477,Z 524.403,A -85,B 0,C 180,E1 -18407.266,E2 -18407.266} C_VEL
LIN {X 0,Y 278.357,Z 528.217,A -85,B 0,C 180,E1 -18410.199,E2 -18410.199} C_VEL
LIN {X 0,Y 278.781,Z 530.536,A -85,B 0,C 180,E1 -18411.398,E2 -18411.398} C_VEL
LIN {X 0,Y 279.19,Z 535.223,A -85,B 0,C 180,E1 -18413.186,E2 -18413.186} C_VEL
LIN {X 0,Y 279.369,Z 539.859,A -85,B 0,C 180,E1 -18414.647,E2 -18414.647} C_VEL
LIN {X 0,Y 278.859,Z 548.376,A -85,B 0,C 180,E1 -18416.828,E2 -18416.828} C_VEL
LIN {X 0,Y 277.703,Z 558.318,A -85,B 0,C 180,E1 -18419.172,E2 -18419.172} C_VEL
LIN {X 0,Y 275.813,Z 568.287,A -85,B 0,C 180,E1 -18421.46,E2 -18421.46} C_VEL
LIN {X 0,Y 273.376,Z 576.223,A -85,B 0,C 180,E1 -18423.263,E2 -18423.263} C_VEL
LIN {X 0,Y 270.166,Z 583.579,A -85,B 0,C 180,E1 -18424.993,E2 -18424.993} C_VEL
LIN {X 0,Y 265.817,Z 592.47,A -85,B 0,C 180,E1 -18427.457,E2 -18427.457} C_VEL
LIN {X 0,Y 262.566,Z 598.782,A -85,B 0,C 180,E1 -18429.637,E2 -18429.637} C_VEL
LIN {X 0,Y 260.079,Z 604.054,A -85,B 0,C 180,E1 -18431.895,E2 -18431.895} C_VEL
LIN {X 0,Y 257.95,Z 608.337,A -85,B 0,C 180,E1 -18434.189,E2 -18434.189} C_VEL
LIN {X 0,Y 256.682,Z 610.734,A -85,B 0,C 180,E1 -18435.734,E2 -18435.734} C_VEL
LIN {X 0,Y 255.11,Z 614.278,A -85,B 0,C 180,E1 -18438.881,E2 -18438.881} C_VEL
LIN {X 0,Y 254.322,Z 616.35,A -85,B 0,C 180,E1 -18442.058,E2 -18442.058} C_VEL
LIN {X 0,Y 254.205,Z 616.896,A -85,B 0,C 180,E1 -18444.437,E2 -18444.437} C_VEL
LIN {X 0,Y 254.27,Z 616.569,A -85,B 0,C 180,E1 -18446.831,E2 -18446.831} C_VEL
LIN {X 0,Y 254.685,Z 615.525,A -85,B 0,C 180,E1 -18449.209,E2 -18449.209} C_VEL
LIN {X 0,Y 254.457,Z 617.349,A -85,B 0,C 180,E1 -18451.583,E2 -18451.583} C_VEL
LIN {X 0,Y 254.16,Z 618.359,A -85,B 0,C 180,E1 -18454.758,E2 -18454.758} C_VEL
LIN {X 0,Y 254.15,Z 618.278,A -85,B 0,C 180,E1 -18456.351,E2 -18456.351} C_VEL
LIN {X 0,Y 254.634,Z 616.942,A -85,B 0,C 180,E1 -18459.532,E2 -18459.532} C_VEL
LIN {X 0,Y 255.784,Z 614.14,A -85,B 0,C 180,E1 -18462.698,E2 -18462.698} C_VEL
LIN {X 0,Y 257.29,Z 611.058,A -85,B 0,C 180,E1 -18465.04,E2 -18465.04} C_VEL
LIN {X 0,Y 260.034,Z 605.581,A -85,B 0,C 180,E1 -18468.108,E2 -18468.108} C_VEL
LIN {X 0,Y 263.546,Z 598.43,A -85,B 0,C 180,E1 -18471.1,E2 -18471.1} C_VEL
LIN {X 0,Y 267.574,Z 590.587,A -85,B 0,C 180,E1 -18473.613,E2 -18473.613} C_VEL
LIN {X 0,Y 272.272,Z 581.103,A -85,B 0,C 180,E1 -18476.028,E2 -18476.028} C_VEL
LIN {X 0,Y 275.317,Z 573.348,A -85,B 0,C 180,E1 -18477.766,E2 -18477.766} C_VEL
LIN {X 0,Y 276.862,Z 566.912,A -85,B 0,C 180,E1 -18479.285,E2 -18479.285} C_VEL
LIN {X 0,Y 277.967,Z 557.425,A -85,B 0,C 180,E1 -18481.643,E2 -18481.643} C_VEL
LIN {X 0,Y 278.17,Z 549.642,A -85,B 0,C 180,E1 -18483.768,E2 -18483.768} C_VEL
LIN {X 0,Y 277.956,Z 542.465,A -85,B 0,C 180,E1 -18485.992,E2 -18485.992} C_VEL
LIN {X 0,Y 277.574,Z 537.472,A -85,B 0,C 180,E1 -18487.833,E2 -18487.833} C_VEL
LIN {X 0,Y 277.27,Z 534.04,A -85,B 0,C 180,E1 -18489.322,E2 -18489.322} C_VEL
LIN {X 0,Y 276.366,Z 529.52,A -85,B 0,C 180,E1 -18492.484,E2 -18492.484} C_VEL
LIN {X 0,Y 276.342,Z 528.381,A -85,B 0,C 180,E1 -18493.367,E2 -18493.367} C_VEL
LIN {X 0,Y 276.3,Z 526.924,A -85,B 0,C 180,E1 -18495.415,E2 -18495.415} C_VEL
LIN {X 0,Y 276.299,Z 526.884,A -85,B 0,C 180,E1 -18497.532,E2 -18497.532} C_VEL
LIN {X 0,Y 277.236,Z 528.116,A -85,B 0,C 180,E1 -18500.672,E2 -18500.672} C_VEL
LIN {X 0,Y 278.283,Z 529.719,A -85,B 0,C 180,E1 -18502.691,E2 -18502.691} C_VEL
LIN {X 0,Y 279.416,Z 532.253,A -85,B 0,C 180,E1 -18504.655,E2 -18504.655} C_VEL
LIN {X 0,Y 280.841,Z 536.948,A -85,B 0,C 180,E1 -18507.196,E2 -18507.196} C_VEL
LIN {X 0,Y 281.851,Z 541.841,A -85,B 0,C 180,E1 -18509.286,E2 -18509.286} C_VEL
LIN {X 0,Y 282.419,Z 547.584,A -85,B 0,C 180,E1 -18511.39,E2 -18511.39} C_VEL
LIN {X 0,Y 282.451,Z 548.779,A -85,B 0,C 180,E1 -18511.787,E2 -18511.787} C_VEL
LIN {X 0,Y 282.004,Z 550.422,A -85,B 0,C 180,E1 -18512.187,E2 -18512.187} C_VEL
LIN {X 0,Y 276.842,Z 560.99,A -85,B 0,C 180,E1 -18514.433,E2 -18514.433} C_VEL
LIN {X 0,Y 272.1,Z 569.703,A -85,B 0,C 180,E1 -18516.804,E2 -18516.804} C_VEL
LIN {X 0,Y 267.912,Z 576.772,A -85,B 0,C 180,E1 -18519.26,E2 -18519.26} C_VEL
LIN {X 0,Y 263.939,Z 582.976,A -85,B 0,C 180,E1 -18522.169,E2 -18522.169} C_VEL
LIN {X 0,Y 261.459,Z 586.536,A -85,B 0,C 180,E1 -18524.407,E2 -18524.407} C_VEL
LIN {X 0,Y 259.922,Z 588.446,A -85,B 0,C 180,E1 -18525.916,E2 -18525.916} C_VEL
LIN {X 0,Y 257.704,Z 591.022,A -85,B 0,C 180,E1 -18528.995,E2 -18528.995} C_VEL
LIN {X 0,Y 255.892,Z 592.147,A -85,B 0,C 180,E1 -18532.107,E2 -18532.107} C_VEL
LIN {X 0,Y 255.038,Z 591.768,A -85,B 0,C 180,E1 -18535.258,E2 -18535.258} C_VEL
LIN {X 0,Y 254.418,Z 589.833,A -85,B 0,C 180,E1 -18538.417,E2 -18538.417} C_VEL
LIN {X 0,Y 254.266,Z 586.343,A -85,B 0,C 180,E1 -18541.584,E2 -18541.584} C_VEL
LIN {X 0,Y 254.375,Z 582.588,A -85,B 0,C 180,E1 -18543.961,E2 -18543.961} C_VEL
LIN {X 0,Y 254.566,Z 577.765,A -85,B 0,C 180,E1 -18546.341,E2 -18546.341} C_VEL
LIN {X 0,Y 254.998,Z 571.705,A -85,B 0,C 180,E1 -18548.719,E2 -18548.719} C_VEL
LIN {X 0,Y 255.637,Z 564.24,A -85,B 0,C 180,E1 -18551.096,E2 -18551.096} C_VEL
LIN {X 0,Y 256.559,Z 555.146,A -85,B 0,C 180,E1 -18553.465,E2 -18553.465} C_VEL
LIN {X 0,Y 257.746,Z 544.935,A -85,B 0,C 180,E1 -18555.621,E2 -18555.621} C_VEL
LIN {X 0,Y 258.946,Z 534.883,A -85,B 0,C 180,E1 -18557.371,E2 -18557.371} C_VEL
LIN {X 0,Y 259.935,Z 524.087,A -85,B 0,C 180,E1 -18558.933,E2 -18558.933} C_VEL
LIN {X 0,Y 260.445,Z 517.736,A -85,B 0,C 180,E1 -18559.713,E2 -18559.713} C_VEL
LIN {X 0,Y 257.878,Z 503.904,A -85,B 0,C 180,E1 -18561.236,E2 -18561.236} C_VEL
LIN {X 0,Y 255.296,Z 489.754,A -85,B 0,C 180,E1 -18562.437,E2 -18562.437} C_VEL
LIN {X 0,Y 254.665,Z 485.724,A -85,B 0,C 180,E1 -18562.729,E2 -18562.729} C_VEL
LIN {X 0,Y 254.732,Z 484.763,A -85,B 0,C 180,E1 -18564.014,E2 -18564.014} C_VEL
LIN {X 0,Y 255.214,Z 484.697,A -85,B 0,C 180,E1 -18568.211,E2 -18568.211} C_VEL
LIN {X 0,Y 255.556,Z 484.648,A -85,B 0,C 180,E1 -18571.512,E2 -18571.512} C_VEL
LIN {X 0,Y 255.88,Z 484.609,A -85,B 0,C 180,E1 -18575.226,E2 -18575.226} C_VEL
LIN {X 0,Y 256.049,Z 484.588,A -85,B 0,C 180,E1 -18579.147,E2 -18579.147} C_VEL
LIN {X 0,Y 256.065,Z 484.585,A -85,B 0,C 180,E1 -18583.327,E2 -18583.327} C_VEL
LIN {X 0,Y 256.075,Z 484.586,A -85,B 0,C 180,E1 -18587.819,E2 -18587.819} C_VEL
LIN {X 0,Y 256.092,Z 484.581,A -85,B 0,C 180,E1 -18590.861,E2 -18590.861} C_VEL
LIN {X 0,Y 256.125,Z 484.579,A -85,B 0,C 180,E1 -18594.814,E2 -18594.814} C_VEL
LIN {X 0,Y 256.097,Z 484.581,A -85,B 0,C 180,E1 -18598.573,E2 -18598.573} C_VEL
LIN {X 0,Y 256.144,Z 484.58,A -85,B 0,C 180,E1 -18602.196,E2 -18602.196} C_VEL
LIN {X 0,Y 256.172,Z 484.574,A -85,B 0,C 180,E1 -18605.699,E2 -18605.699} C_VEL
LIN {X 0,Y 256.171,Z 484.571,A -85,B 0,C 180,E1 -18609.105,E2 -18609.105} C_VEL
LIN {X 0,Y 256.305,Z 484.56,A -85,B 0,C 180,E1 -18614.085,E2 -18614.085} C_VEL
LIN {X 0,Y 256.314,Z 484.554,A -85,B 0,C 180,E1 -18618.934,E2 -18618.934} C_VEL
LIN {X 0,Y 256.545,Z 484.53,A -85,B 0,C 180,E1 -18622.127,E2 -18622.127} C_VEL
LIN {X 0,Y 256.719,Z 484.506,A -85,B 0,C 180,E1 -18628.431,E2 -18628.431} C_VEL
LIN {X 0,Y 256.718,Z 484.506,A -85,B 0,C 180,E1 -18631.569,E2 -18631.569} C_VEL
LIN {X 0,Y 256.468,Z 484.537,A -85,B 0,C 180,E1 -18636.293,E2 -18636.293} C_VEL
LIN {X 0,Y 256.431,Z 484.542,A -85,B 0,C 180,E1 -18639.465,E2 -18639.465} C_VEL
LIN {X 0,Y 256.26,Z 484.563,A -85,B 0,C 180,E1 -18644.29,E2 -18644.29} C_VEL
LIN {X 0,Y 256.215,Z 484.569,A -85,B 0,C 180,E1 -18647.562,E2 -18647.562} C_VEL
LIN {X 0,Y 256.16,Z 484.573,A -85,B 0,C 180,E1 -18651.119,E2 -18651.119} C_VEL
LIN {X 0,Y 256.192,Z 484.57,A -85,B 0,C 180,E1 -18655.138,E2 -18655.138} C_VEL
LIN {X 0,Y 256.115,Z 484.582,A -85,B 0,C 180,E1 -18659.6,E2 -18659.6} C_VEL
LIN {X 0,Y 256.089,Z 484.583,A -85,B 0,C 180,E1 -18663.29,E2 -18663.29} C_VEL
LIN {X 0,Y 256.132,Z 484.578,A -85,B 0,C 180,E1 -18667.275,E2 -18667.275} C_VEL
LIN {X 0,Y 256.06,Z 484.586,A -85,B 0,C 180,E1 -18671.203,E2 -18671.203} C_VEL
LIN {X 0,Y 256.061,Z 484.589,A -85,B 0,C 180,E1 -18675.53,E2 -18675.53} C_VEL
LIN {X 0,Y 256.057,Z 484.585,A -85,B 0,C 180,E1 -18678.796,E2 -18678.796} C_VEL
LIN {X 0,Y 256.069,Z 484.586,A -85,B 0,C 180,E1 -18682.856,E2 -18682.856} C_VEL
LIN {X 0,Y 255.84,Z 484.612,A -85,B 0,C 180,E1 -18686.673,E2 -18686.673} C_VEL
LIN {X 0,Y 255.42,Z 484.667,A -85,B 0,C 180,E1 -18690.311,E2 -18690.311} C_VEL
LIN {X 0,Y 255.003,Z 484.72,A -85,B 0,C 180,E1 -18693.834,E2 -18693.834} C_VEL
LIN {X 0,Y 254.586,Z 484.775,A -85,B 0,C 180,E1 -18697.448,E2 -18697.448} C_VEL
LIN {X 0,Y 257.288,Z 500.675,A -85,B 0,C 180,E1 -18698.711,E2 -18698.711} C_VEL
LIN {X 0,Y 259.762,Z 514.324,A -85,B 0,C 180,E1 -18700.13,E2 -18700.13} C_VEL
LIN {X 0,Y 260.321,Z 518.986,A -85,B 0,C 180,E1 -18700.687,E2 -18700.687} C_VEL
LIN {X 0,Y 259.152,Z 531.013,A -85,B 0,C 180,E1 -18702.291,E2 -18702.291} C_VEL
LIN {X 0,Y 257.901,Z 542.474,A -85,B 0,C 180,E1 -18704.186,E2 -18704.186} C_VEL
LIN {X 0,Y 256.753,Z 552.161,A -85,B 0,C 180,E1 -18706.142,E2 -18706.142} C_VEL
LIN {X 0,Y 255.776,Z 561.762,A -85,B 0,C 180,E1 -18708.509,E2 -18708.509} C_VEL
LIN {X 0,Y 255.076,Z 569.609,A -85,B 0,C 180,E1 -18710.884,E2 -18710.884} C_VEL
LIN {X 0,Y 254.533,Z 576.893,A -85,B 0,C 180,E1 -18713.659,E2 -18713.659} C_VEL
LIN {X 0,Y 254.369,Z 581.798,A -85,B 0,C 180,E1 -18716.039,E2 -18716.039} C_VEL
LIN {X 0,Y 254.243,Z 585.616,A -85,B 0,C 180,E1 -18718.416,E2 -18718.416} C_VEL
LIN {X 0,Y 254.248,Z 587.629,A -85,B 0,C 180,E1 -18720,E2 -18720} C_VEL
LIN {X 0,Y 254.652,Z 590.368,A -85,B 0,C 180,E1 -18723.164,E2 -18723.164} C_VEL
LIN {X 0,Y 254.96,Z 591.164,A -85,B 0,C 180,E1 -18724.743,E2 -18724.743} C_VEL
LIN {X 0,Y 255.317,Z 591.577,A -85,B 0,C 180,E1 -18726.321,E2 -18726.321} C_VEL
LIN {X 0,Y 256.654,Z 591.209,A -85,B 0,C 180,E1 -18729.456,E2 -18729.456} C_VEL
LIN {X 0,Y 257.613,Z 590.473,A -85,B 0,C 180,E1 -18731.009,E2 -18731.009} C_VEL
LIN {X 0,Y 258.502,Z 589.413,A -85,B 0,C 180,E1 -18732.562,E2 -18732.562} C_VEL
LIN {X 0,Y 261.304,Z 586.002,A -85,B 0,C 180,E1 -18735.602,E2 -18735.602} C_VEL
LIN {X 0,Y 263.722,Z 582.442,A -85,B 0,C 180,E1 -18737.846,E2 -18737.846} C_VEL
LIN {X 0,Y 266.685,Z 577.903,A -85,B 0,C 180,E1 -18740.035,E2 -18740.035} C_VEL
LIN {X 0,Y 270.588,Z 571.288,A -85,B 0,C 180,E1 -18742.526,E2 -18742.526} C_VEL
LIN {X 0,Y 274.462,Z 564.339,A -85,B 0,C 180,E1 -18744.589,E2 -18744.589} C_VEL
LIN {X 0,Y 279.446,Z 554.405,A -85,B 0,C 180,E1 -18746.917,E2 -18746.917} C_VEL
LIN {X 0,Y 282.503,Z 547.615,A -85,B 0,C 180,E1 -18748.248,E2 -18748.248} C_VEL
LIN {X 0,Y 282.494,Z 545.567,A -85,B 0,C 180,E1 -18748.923,E2 -18748.923} C_VEL
LIN {X 0,Y 281.572,Z 543.299,A -85,B 0,C 180,E1 -18750.015,E2 -18750.015} C_VEL
LIN {X 0,Y 278.901,Z 540.788,A -85,B 0,C 180,E1 -18751.931,E2 -18751.931} C_VEL
LIN {X 0,Y 276.675,Z 538.156,A -85,B 0,C 180,E1 -18753.91,E2 -18753.91} C_VEL
LIN {X 0,Y 276.48,Z 537.436,A -85,B 0,C 180,E1 -18754.302,E2 -18754.302} C_VEL
LIN {X 0,Y 275.902,Z 534.658,A -85,B 0,C 180,E1 -18755.865,E2 -18755.865} C_VEL
LIN {X 0,Y 275.111,Z 532.063,A -85,B 0,C 180,E1 -18757.814,E2 -18757.814} C_VEL
LIN {X 0,Y 274.334,Z 530.345,A -85,B 0,C 180,E1 -18759.826,E2 -18759.826} C_VEL
LIN {X 0,Y 273.898,Z 529.251,A -85,B 0,C 180,E1 -18761.916,E2 -18761.916} C_VEL
LIN {X 0,Y 273.807,Z 528.914,A -85,B 0,C 180,E1 -18764.053,E2 -18764.053} C_VEL
LIN {X 0,Y 273.866,Z 529.819,A -85,B 0,C 180,E1 -18766.141,E2 -18766.141} C_VEL
LIN {X 0,Y 274.131,Z 531.842,A -85,B 0,C 180,E1 -18768.197,E2 -18768.197} C_VEL
LIN {X 0,Y 274.756,Z 534.645,A -85,B 0,C 180,E1 -18770.247,E2 -18770.247} C_VEL
LIN {X 0,Y 274.965,Z 538.951,A -85,B 0,C 180,E1 -18772.162,E2 -18772.162} C_VEL
LIN {X 0,Y 274.85,Z 544.25,A -85,B 0,C 180,E1 -18773.976,E2 -18773.976} C_VEL
LIN {X 0,Y 273.9,Z 552.237,A -85,B 0,C 180,E1 -18776.147,E2 -18776.147} C_VEL
LIN {X 0,Y 272.401,Z 561.062,A -85,B 0,C 180,E1 -18778.365,E2 -18778.365} C_VEL
LIN {X 0,Y 270.033,Z 570.905,A -85,B 0,C 180,E1 -18780.791,E2 -18780.791} C_VEL
LIN {X 0,Y 267.33,Z 578.404,A -85,B 0,C 180,E1 -18782.608,E2 -18782.608} C_VEL
LIN {X 0,Y 262.554,Z 587.912,A -85,B 0,C 180,E1 -18785.065,E2 -18785.065} C_VEL
LIN {X 0,Y 258.255,Z 595.838,A -85,B 0,C 180,E1 -18787.605,E2 -18787.605} C_VEL
LIN {X 0,Y 255.083,Z 601.49,A -85,B 0,C 180,E1 -18789.855,E2 -18789.855} C_VEL
LIN {X 0,Y 251.873,Z 607.448,A -85,B 0,C 180,E1 -18792.963,E2 -18792.963} C_VEL
LIN {X 0,Y 249.813,Z 610.907,A -85,B 0,C 180,E1 -18795.333,E2 -18795.333} C_VEL
LIN {X 0,Y 248.12,Z 614.197,A -85,B 0,C 180,E1 -18798.564,E2 -18798.564} C_VEL
LIN {X 0,Y 247.266,Z 616.006,A -85,B 0,C 180,E1 -18801.83,E2 -18801.83} C_VEL
LIN {X 0,Y 247.137,Z 616.297,A -85,B 0,C 180,E1 -18805.106,E2 -18805.106} C_VEL
LIN {X 0,Y 247.537,Z 615.087,A -85,B 0,C 180,E1 -18808.373,E2 -18808.373} C_VEL
LIN {X 0,Y 247.67,Z 614.548,A -85,B 0,C 180,E1 -18809.187,E2 -18809.187} C_VEL
LIN {X 0,Y 247.411,Z 616.559,A -85,B 0,C 180,E1 -18811.628,E2 -18811.628} C_VEL
LIN {X 0,Y 247.081,Z 617.744,A -85,B 0,C 180,E1 -18814.895,E2 -18814.895} C_VEL
LIN {X 0,Y 247.25,Z 617.429,A -85,B 0,C 180,E1 -18818.171,E2 -18818.171} C_VEL
LIN {X 0,Y 248.136,Z 615.62,A -85,B 0,C 180,E1 -18821.435,E2 -18821.435} C_VEL
LIN {X 0,Y 249.813,Z 612.35,A -85,B 0,C 180,E1 -18824.667,E2 -18824.667} C_VEL
LIN {X 0,Y 252.564,Z 607.6,A -85,B 0,C 180,E1 -18827.824,E2 -18827.824} C_VEL
LIN {X 0,Y 255.379,Z 602.326,A -85,B 0,C 180,E1 -18830.46,E2 -18830.46} C_VEL
LIN {X 0,Y 259.914,Z 594.28,A -85,B 0,C 180,E1 -18833.506,E2 -18833.506} C_VEL
LIN {X 0,Y 264.644,Z 585.758,A -85,B 0,C 180,E1 -18835.988,E2 -18835.988} C_VEL
LIN {X 0,Y 268.195,Z 578.729,A -85,B 0,C 180,E1 -18837.719,E2 -18837.719} C_VEL
LIN {X 0,Y 270.383,Z 572.729,A -85,B 0,C 180,E1 -18839.168,E2 -18839.168} C_VEL
LIN {X 0,Y 271.993,Z 565.278,A -85,B 0,C 180,E1 -18841.116,E2 -18841.116} C_VEL
LIN {X 0,Y 272.925,Z 557.859,A -85,B 0,C 180,E1 -18843.151,E2 -18843.151} C_VEL
LIN {X 0,Y 273.345,Z 550.436,A -85,B 0,C 180,E1 -18845.436,E2 -18845.436} C_VEL
LIN {X 0,Y 273.395,Z 543.163,A -85,B 0,C 180,E1 -18848.094,E2 -18848.094} C_VEL
LIN {X 0,Y 273.168,Z 539.138,A -85,B 0,C 180,E1 -18850.031,E2 -18850.031} C_VEL
LIN {X 0,Y 272.702,Z 535.18,A -85,B 0,C 180,E1 -18852.963,E2 -18852.963} C_VEL
LIN {X 0,Y 272.739,Z 534,A -85,B 0,C 180,E1 -18854.087,E2 -18854.087} C_VEL
LIN {X 0,Y 272.753,Z 532.97,A -85,B 0,C 180,E1 -18856.176,E2 -18856.176} C_VEL
LIN {X 0,Y 272.816,Z 533.292,A -85,B 0,C 180,E1 -18858.337,E2 -18858.337} C_VEL
LIN {X 0,Y 273.422,Z 534.055,A -85,B 0,C 180,E1 -18860.454,E2 -18860.454} C_VEL
LIN {X 0,Y 274.345,Z 535.615,A -85,B 0,C 180,E1 -18862.574,E2 -18862.574} C_VEL
LIN {X 0,Y 275.325,Z 538.379,A -85,B 0,C 180,E1 -18864.77,E2 -18864.77} C_VEL
LIN {X 0,Y 276.55,Z 543.817,A -85,B 0,C 180,E1 -18867.746,E2 -18867.746} C_VEL
LIN {X 0,Y 277.033,Z 549.821,A -85,B 0,C 180,E1 -18870.255,E2 -18870.255} C_VEL
LIN {X 0,Y 276.976,Z 552.269,A -85,B 0,C 180,E1 -18871.177,E2 -18871.177} C_VEL
LIN {X 0,Y 272.393,Z 561.261,A -85,B 0,C 180,E1 -18873.159,E2 -18873.159} C_VEL
LIN {X 0,Y 267.257,Z 569.948,A -85,B 0,C 180,E1 -18875.533,E2 -18875.533} C_VEL
LIN {X 0,Y 262.69,Z 577.047,A -85,B 0,C 180,E1 -18878.003,E2 -18878.003} C_VEL
LIN {X 0,Y 258.314,Z 583.287,A -85,B 0,C 180,E1 -18880.945,E2 -18880.945} C_VEL
LIN {X 0,Y 254.756,Z 587.903,A -85,B 0,C 180,E1 -18883.986,E2 -18883.986} C_VEL
LIN {X 0,Y 253.142,Z 589.607,A -85,B 0,C 180,E1 -18885.531,E2 -18885.531} C_VEL
LIN {X 0,Y 250.683,Z 591.997,A -85,B 0,C 180,E1 -18888.885,E2 -18888.885} C_VEL
LIN {X 0,Y 248.909,Z 592.762,A -85,B 0,C 180,E1 -18891.884,E2 -18891.884} C_VEL
LIN {X 0,Y 247.982,Z 592.081,A -85,B 0,C 180,E1 -18895.123,E2 -18895.123} C_VEL
LIN {X 0,Y 247.34,Z 589.933,A -85,B 0,C 180,E1 -18898.372,E2 -18898.372} C_VEL
LIN {X 0,Y 247.172,Z 587.269,A -85,B 0,C 180,E1 -18900.815,E2 -18900.815} C_VEL
LIN {X 0,Y 247.243,Z 583.637,A -85,B 0,C 180,E1 -18903.259,E2 -18903.259} C_VEL
LIN {X 0,Y 247.346,Z 579.409,A -85,B 0,C 180,E1 -18905.491,E2 -18905.491} C_VEL
LIN {X 0,Y 247.832,Z 573.131,A -85,B 0,C 180,E1 -18908.152,E2 -18908.152} C_VEL
LIN {X 0,Y 248.42,Z 565.958,A -85,B 0,C 180,E1 -18910.597,E2 -18910.597} C_VEL
LIN {X 0,Y 249.297,Z 557.139,A -85,B 0,C 180,E1 -18913.035,E2 -18913.035} C_VEL
LIN {X 0,Y 250.271,Z 548.263,A -85,B 0,C 180,E1 -18915.056,E2 -18915.056} C_VEL
LIN {X 0,Y 251.476,Z 537.592,A -85,B 0,C 180,E1 -18917.065,E2 -18917.065} C_VEL
LIN {X 0,Y 252.557,Z 526.959,A -85,B 0,C 180,E1 -18918.706,E2 -18918.706} C_VEL
LIN {X 0,Y 253.274,Z 517.987,A -85,B 0,C 180,E1 -18919.873,E2 -18919.873} C_VEL
LIN {X 0,Y 250.86,Z 504.934,A -85,B 0,C 180,E1 -18921.359,E2 -18921.359} C_VEL
LIN {X 0,Y 248.38,Z 491.18,A -85,B 0,C 180,E1 -18922.587,E2 -18922.587} C_VEL
LIN {X 0,Y 247.609,Z 486.118,A -85,B 0,C 180,E1 -18922.972,E2 -18922.972} C_VEL
LIN {X 0,Y 247.66,Z 485.643,A -85,B 0,C 180,E1 -18923.808,E2 -18923.808} C_VEL
LIN {X 0,Y 248.191,Z 485.569,A -85,B 0,C 180,E1 -18928.618,E2 -18928.618} C_VEL
LIN {X 0,Y 248.569,Z 485.521,A -85,B 0,C 180,E1 -18932.494,E2 -18932.494} C_VEL
LIN {X 0,Y 248.885,Z 485.484,A -85,B 0,C 180,E1 -18936.371,E2 -18936.371} C_VEL
LIN {X 0,Y 248.991,Z 485.469,A -85,B 0,C 180,E1 -18940.35,E2 -18940.35} C_VEL
LIN {X 0,Y 249.012,Z 485.464,A -85,B 0,C 180,E1 -18942.793,E2 -18942.793} C_VEL
LIN {X 0,Y 249.019,Z 485.464,A -85,B 0,C 180,E1 -18947.363,E2 -18947.363} C_VEL
LIN {X 0,Y 249.042,Z 485.46,A -85,B 0,C 180,E1 -18951.622,E2 -18951.622} C_VEL
LIN {X 0,Y 249.065,Z 485.459,A -85,B 0,C 180,E1 -18955.643,E2 -18955.643} C_VEL
LIN {X 0,Y 249.055,Z 485.457,A -85,B 0,C 180,E1 -18959.473,E2 -18959.473} C_VEL
LIN {X 0,Y 249.077,Z 485.457,A -85,B 0,C 180,E1 -18963.163,E2 -18963.163} C_VEL
LIN {X 0,Y 249.084,Z 485.455,A -85,B 0,C 180,E1 -18966.733,E2 -18966.733} C_VEL
LIN {X 0,Y 249.116,Z 485.455,A -85,B 0,C 180,E1 -18970.212,E2 -18970.212} C_VEL
LIN {X 0,Y 249.246,Z 485.437,A -85,B 0,C 180,E1 -18973.622,E2 -18973.622} C_VEL
LIN {X 0,Y 249.258,Z 485.434,A -85,B 0,C 180,E1 -18978.617,E2 -18978.617} C_VEL
LIN {X 0,Y 249.489,Z 485.409,A -85,B 0,C 180,E1 -18981.903,E2 -18981.903} C_VEL
LIN {X 0,Y 249.441,Z 485.41,A -85,B 0,C 180,E1 -18986.77,E2 -18986.77} C_VEL
LIN {X 0,Y 249.733,Z 485.379,A -85,B 0,C 180,E1 -18990,E2 -18990} C_VEL
LIN {X 0,Y 249.436,Z 485.411,A -85,B 0,C 180,E1 -18993.23,E2 -18993.23} C_VEL
LIN {X 0,Y 249.441,Z 485.412,A -85,B 0,C 180,E1 -18996.471,E2 -18996.471} C_VEL
LIN {X 0,Y 249.348,Z 485.426,A -85,B 0,C 180,E1 -18999.736,E2 -18999.736} C_VEL
LIN {X 0,Y 249.21,Z 485.439,A -85,B 0,C 180,E1 -19004.703,E2 -19004.703} C_VEL
LIN {X 0,Y 249.144,Z 485.451,A -85,B 0,C 180,E1 -19008.077,E2 -19008.077} C_VEL
LIN {X 0,Y 249.091,Z 485.455,A -85,B 0,C 180,E1 -19011.518,E2 -19011.518} C_VEL
LIN {X 0,Y 249.134,Z 485.451,A -85,B 0,C 180,E1 -19015.482,E2 -19015.482} C_VEL
LIN {X 0,Y 249.084,Z 485.455,A -85,B 0,C 180,E1 -19018.992,E2 -19018.992} C_VEL
LIN {X 0,Y 249.04,Z 485.461,A -85,B 0,C 180,E1 -19022.425,E2 -19022.425} C_VEL
LIN {X 0,Y 249.073,Z 485.458,A -85,B 0,C 180,E1 -19026.338,E2 -19026.338} C_VEL
LIN {X 0,Y 249.029,Z 485.461,A -85,B 0,C 180,E1 -19030.474,E2 -19030.474} C_VEL
LIN {X 0,Y 249.006,Z 485.465,A -85,B 0,C 180,E1 -19034.879,E2 -19034.879} C_VEL
LIN {X 0,Y 249.019,Z 485.464,A -85,B 0,C 180,E1 -19037.363,E2 -19037.363} C_VEL
LIN {X 0,Y 249.01,Z 485.468,A -85,B 0,C 180,E1 -19041.616,E2 -19041.616} C_VEL
LIN {X 0,Y 248.854,Z 485.487,A -85,B 0,C 180,E1 -19045.609,E2 -19045.609} C_VEL
LIN {X 0,Y 248.495,Z 485.53,A -85,B 0,C 180,E1 -19049.397,E2 -19049.397} C_VEL
LIN {X 0,Y 248.06,Z 485.584,A -85,B 0,C 180,E1 -19053.043,E2 -19053.043} C_VEL
LIN {X 0,Y 247.578,Z 485.652,A -85,B 0,C 180,E1 -19057.246,E2 -19057.246} C_VEL
LIN {X 0,Y 250.003,Z 500.009,A -85,B 0,C 180,E1 -19058.423,E2 -19058.423} C_VEL
LIN {X 0,Y 252.383,Z 513.508,A -85,B 0,C 180,E1 -19059.842,E2 -19059.842} C_VEL
LIN {X 0,Y 253.238,Z 519.268,A -85,B 0,C 180,E1 -19060.547,E2 -19060.547} C_VEL
LIN {X 0,Y 252.105,Z 530.968,A -85,B 0,C 180,E1 -19062.142,E2 -19062.142} C_VEL
LIN {X 0,Y 250.772,Z 542.784,A -85,B 0,C 180,E1 -19064.142,E2 -19064.142} C_VEL
LIN {X 0,Y 249.626,Z 552.501,A -85,B 0,C 180,E1 -19066.154,E2 -19066.154} C_VEL
LIN {X 0,Y 248.646,Z 562.101,A -85,B 0,C 180,E1 -19068.588,E2 -19068.588} C_VEL
LIN {X 0,Y 247.948,Z 569.92,A -85,B 0,C 180,E1 -19071.031,E2 -19071.031} C_VEL
LIN {X 0,Y 247.405,Z 577.112,A -85,B 0,C 180,E1 -19073.85,E2 -19073.85} C_VEL
LIN {X 0,Y 247.238,Z 582.879,A -85,B 0,C 180,E1 -19076.74,E2 -19076.74} C_VEL
LIN {X 0,Y 247.145,Z 586.568,A -85,B 0,C 180,E1 -19079.185,E2 -19079.185} C_VEL
LIN {X 0,Y 247.302,Z 589.268,A -85,B 0,C 180,E1 -19081.628,E2 -19081.628} C_VEL
LIN {X 0,Y 247.583,Z 590.554,A -85,B 0,C 180,E1 -19083.254,E2 -19083.254} C_VEL
LIN {X 0,Y 248.272,Z 592,A -85,B 0,C 180,E1 -19086.501,E2 -19086.501} C_VEL
LIN {X 0,Y 248.842,Z 592.172,A -85,B 0,C 180,E1 -19088.118,E2 -19088.118} C_VEL
LIN {X 0,Y 250.709,Z 591.328,A -85,B 0,C 180,E1 -19091.316,E2 -19091.316} C_VEL
LIN {X 0,Y 251.647,Z 590.387,A -85,B 0,C 180,E1 -19092.91,E2 -19092.91} C_VEL
LIN {X 0,Y 254.612,Z 587.34,A -85,B 0,C 180,E1 -19096.023,E2 -19096.023} C_VEL
LIN {X 0,Y 257.159,Z 584.057,A -85,B 0,C 180,E1 -19098.318,E2 -19098.318} C_VEL
LIN {X 0,Y 261.349,Z 578.149,A -85,B 0,C 180,E1 -19101.286,E2 -19101.286} C_VEL
LIN {X 0,Y 265.63,Z 571.543,A -85,B 0,C 180,E1 -19103.796,E2 -19103.796} C_VEL
LIN {X 0,Y 270.554,Z 563.245,A -85,B 0,C 180,E1 -19106.206,E2 -19106.206} C_VEL
LIN {X 0,Y 275.174,Z 554.666,A -85,B 0,C 180,E1 -19108.196,E2 -19108.196} C_VEL
LIN {X 0,Y 277.069,Z 550.563,A -85,B 0,C 180,E1 -19109.064,E2 -19109.064} C_VEL
LIN {X 0,Y 277.351,Z 548.784,A -85,B 0,C 180,E1 -19109.613,E2 -19109.613} C_VEL
LIN {X 0,Y 277.248,Z 543.815,A -85,B 0,C 180,E1 -19111.469,E2 -19111.469} C_VEL
LIN {X 0,Y 276.594,Z 538.059,A -85,B 0,C 180,E1 -19113.986,E2 -19113.986} C_VEL
LIN {X 0,Y 276.48,Z 537.436,A -85,B 0,C 180,E1 -19114.302,E2 -19114.302} C_VEL
LIN {X 0,Y 276.009,Z 536.271,A -85,B 0,C 180,E1 -19115.074,E2 -19115.074} C_VEL
LIN {X 0,Y 275.225,Z 535.654,A -85,B 0,C 180,E1 -19115.867,E2 -19115.867} C_VEL
LIN {X 0,Y 273.207,Z 535.515,A -85,B 0,C 180,E1 -19117.475,E2 -19117.475} C_VEL
LIN {X 0,Y 270.642,Z 536.025,A -85,B 0,C 180,E1 -19119.981,E2 -19119.981} C_VEL
LIN {X 0,Y 270.286,Z 535.82,A -85,B 0,C 180,E1 -19120.832,E2 -19120.832} C_VEL
LIN {X 0,Y 270.152,Z 535.1,A -85,B 0,C 180,E1 -19123.246,E2 -19123.246} C_VEL
LIN {X 0,Y 270.198,Z 535.566,A -85,B 0,C 180,E1 -19125.389,E2 -19125.389} C_VEL
LIN {X 0,Y 270.324,Z 537.236,A -85,B 0,C 180,E1 -19127.471,E2 -19127.471} C_VEL
LIN {X 0,Y 270.677,Z 539.721,A -85,B 0,C 180,E1 -19129.525,E2 -19129.525} C_VEL
LIN {X 0,Y 270.766,Z 541.091,A -85,B 0,C 180,E1 -19130.335,E2 -19130.335} C_VEL
LIN {X 0,Y 270.612,Z 544.835,A -85,B 0,C 180,E1 -19131.962,E2 -19131.962} C_VEL
LIN {X 0,Y 270.291,Z 548.527,A -85,B 0,C 180,E1 -19133.27,E2 -19133.27} C_VEL
LIN {X 0,Y 268.68,Z 557.021,A -85,B 0,C 180,E1 -19135.713,E2 -19135.713} C_VEL
LIN {X 0,Y 267.035,Z 564.26,A -85,B 0,C 180,E1 -19137.653,E2 -19137.653} C_VEL
LIN {X 0,Y 264.282,Z 573.509,A -85,B 0,C 180,E1 -19140.091,E2 -19140.091} C_VEL
LIN {X 0,Y 260.647,Z 581.891,A -85,B 0,C 180,E1 -19142.282,E2 -19142.282} C_VEL
LIN {X 0,Y 254.913,Z 591.792,A -85,B 0,C 180,E1 -19145.137,E2 -19145.137} C_VEL
LIN {X 0,Y 251.178,Z 598.035,A -85,B 0,C 180,E1 -19147.42,E2 -19147.42} C_VEL
LIN {X 0,Y 248.473,Z 602.252,A -85,B 0,C 180,E1 -19149.295,E2 -19149.295} C_VEL
LIN {X 0,Y 245.101,Z 607.892,A -85,B 0,C 180,E1 -19152.478,E2 -19152.478} C_VEL
LIN {X 0,Y 242.962,Z 611.094,A -85,B 0,C 180,E1 -19154.91,E2 -19154.91} C_VEL
LIN {X 0,Y 241.874,Z 612.775,A -85,B 0,C 180,E1 -19156.559,E2 -19156.559} C_VEL
LIN {X 0,Y 240.595,Z 615.014,A -85,B 0,C 180,E1 -19159.906,E2 -19159.906} C_VEL
LIN {X 0,Y 240.074,Z 615.832,A -85,B 0,C 180,E1 -19163.275,E2 -19163.275} C_VEL
LIN {X 0,Y 240.061,Z 615.692,A -85,B 0,C 180,E1 -19164.961,E2 -19164.961} C_VEL
LIN {X 0,Y 240.478,Z 614.192,A -85,B 0,C 180,E1 -19168.325,E2 -19168.325} C_VEL
LIN {X 0,Y 240.65,Z 613.65,A -85,B 0,C 180,E1 -19169.268,E2 -19169.268} C_VEL
LIN {X 0,Y 240.364,Z 615.675,A -85,B 0,C 180,E1 -19171.676,E2 -19171.676} C_VEL
LIN {X 0,Y 240.011,Z 617.117,A -85,B 0,C 180,E1 -19175.04,E2 -19175.04} C_VEL
LIN {X 0,Y 240.199,Z 617.01,A -85,B 0,C 180,E1 -19178.412,E2 -19178.412} C_VEL
LIN {X 0,Y 241.16,Z 615.472,A -85,B 0,C 180,E1 -19181.771,E2 -19181.771} C_VEL
LIN {X 0,Y 242.961,Z 612.508,A -85,B 0,C 180,E1 -19185.09,E2 -19185.09} C_VEL
LIN {X 0,Y 245.823,Z 608.061,A -85,B 0,C 180,E1 -19188.33,E2 -19188.33} C_VEL
LIN {X 0,Y 249.391,Z 602.129,A -85,B 0,C 180,E1 -19191.491,E2 -19191.491} C_VEL
LIN {X 0,Y 253.517,Z 595.546,A -85,B 0,C 180,E1 -19194.136,E2 -19194.136} C_VEL
LIN {X 0,Y 259.194,Z 586.254,A -85,B 0,C 180,E1 -19197.012,E2 -19197.012} C_VEL
LIN {X 0,Y 262.84,Z 579.429,A -85,B 0,C 180,E1 -19198.77,E2 -19198.77} C_VEL
LIN {X 0,Y 265.055,Z 573.833,A -85,B 0,C 180,E1 -19200.251,E2 -19200.251} C_VEL
LIN {X 0,Y 266.793,Z 566.618,A -85,B 0,C 180,E1 -19202.282,E2 -19202.282} C_VEL
LIN {X 0,Y 267.876,Z 560.025,A -85,B 0,C 180,E1 -19204.287,E2 -19204.287} C_VEL
LIN {X 0,Y 268.632,Z 553.001,A -85,B 0,C 180,E1 -19206.662,E2 -19206.662} C_VEL
LIN {X 0,Y 268.96,Z 547.642,A -85,B 0,C 180,E1 -19208.839,E2 -19208.839} C_VEL
LIN {X 0,Y 269.004,Z 546.075,A -85,B 0,C 180,E1 -19209.583,E2 -19209.583} C_VEL
LIN {X 0,Y 268.805,Z 542.931,A -85,B 0,C 180,E1 -19211.624,E2 -19211.624} C_VEL
LIN {X 0,Y 268.803,Z 541.327,A -85,B 0,C 180,E1 -19212.94,E2 -19212.94} C_VEL
LIN {X 0,Y 268.892,Z 539.468,A -85,B 0,C 180,E1 -19215.114,E2 -19215.114} C_VEL
LIN {X 0,Y 268.932,Z 539.038,A -85,B 0,C 180,E1 -19217.199,E2 -19217.199} C_VEL
LIN {X 0,Y 269.114,Z 539.528,A -85,B 0,C 180,E1 -19219.241,E2 -19219.241} C_VEL
LIN {X 0,Y 269.785,Z 540.535,A -85,B 0,C 180,E1 -19221.4,E2 -19221.4} C_VEL
LIN {X 0,Y 270.57,Z 542.624,A -85,B 0,C 180,E1 -19223.632,E2 -19223.632} C_VEL
LIN {X 0,Y 271.257,Z 546.124,A -85,B 0,C 180,E1 -19226.006,E2 -19226.006} C_VEL
LIN {X 0,Y 271.696,Z 550.368,A -85,B 0,C 180,E1 -19228.221,E2 -19228.221} C_VEL
LIN {X 0,Y 271.673,Z 554.666,A -85,B 0,C 180,E1 -19230.087,E2 -19230.087} C_VEL
LIN {X 0,Y 271.415,Z 555.927,A -85,B 0,C 180,E1 -19230.529,E2 -19230.529} C_VEL
LIN {X 0,Y 265.685,Z 565.615,A -85,B 0,C 180,E1 -19232.851,E2 -19232.851} C_VEL
LIN {X 0,Y 260.449,Z 573.554,A -85,B 0,C 180,E1 -19235.276,E2 -19235.276} C_VEL
LIN {X 0,Y 256.383,Z 579.127,A -85,B 0,C 180,E1 -19237.433,E2 -19237.433} C_VEL
LIN {X 0,Y 251.809,Z 584.998,A -85,B 0,C 180,E1 -19240.433,E2 -19240.433} C_VEL
LIN {X 0,Y 248.054,Z 589.202,A -85,B 0,C 180,E1 -19243.542,E2 -19243.542} C_VEL
LIN {X 0,Y 246.381,Z 590.768,A -85,B 0,C 180,E1 -19245.125,E2 -19245.125} C_VEL
LIN {X 0,Y 243.921,Z 592.752,A -85,B 0,C 180,E1 -19248.365,E2 -19248.365} C_VEL
LIN {X 0,Y 241.908,Z 593.3,A -85,B 0,C 180,E1 -19251.648,E2 -19251.648} C_VEL
LIN {X 0,Y 240.93,Z 592.38,A -85,B 0,C 180,E1 -19254.98,E2 -19254.98} C_VEL
LIN {X 0,Y 240.539,Z 591.367,A -85,B 0,C 180,E1 -19256.65,E2 -19256.65} C_VEL
LIN {X 0,Y 240.124,Z 588.134,A -85,B 0,C 180,E1 -19260,E2 -19260} C_VEL
LIN {X 0,Y 240.156,Z 584.651,A -85,B 0,C 180,E1 -19262.516,E2 -19262.516} C_VEL
LIN {X 0,Y 240.24,Z 579.448,A -85,B 0,C 180,E1 -19265.376,E2 -19265.376} C_VEL
LIN {X 0,Y 240.719,Z 573.373,A -85,B 0,C 180,E1 -19267.989,E2 -19267.989} C_VEL
LIN {X 0,Y 241.284,Z 566.179,A -85,B 0,C 180,E1 -19270.489,E2 -19270.489} C_VEL
LIN {X 0,Y 242.167,Z 557.345,A -85,B 0,C 180,E1 -19272.998,E2 -19272.998} C_VEL
LIN {X 0,Y 243.136,Z 548.503,A -85,B 0,C 180,E1 -19275.08,E2 -19275.08} C_VEL
LIN {X 0,Y 244.356,Z 537.889,A -85,B 0,C 180,E1 -19277.146,E2 -19277.146} C_VEL
LIN {X 0,Y 245.274,Z 528.899,A -85,B 0,C 180,E1 -19278.6,E2 -19278.6} C_VEL
LIN {X 0,Y 246.238,Z 519.458,A -85,B 0,C 180,E1 -19279.888,E2 -19279.888} C_VEL
LIN {X 0,Y 243.945,Z 506.529,A -85,B 0,C 180,E1 -19281.428,E2 -19281.428} C_VEL
LIN {X 0,Y 241.476,Z 492.644,A -85,B 0,C 180,E1 -19282.743,E2 -19282.743} C_VEL
LIN {X 0,Y 240.544,Z 486.526,A -85,B 0,C 180,E1 -19283.231,E2 -19283.231} C_VEL
LIN {X 0,Y 241.03,Z 486.465,A -85,B 0,C 180,E1 -19287.81,E2 -19287.81} C_VEL
LIN {X 0,Y 241.519,Z 486.399,A -85,B 0,C 180,E1 -19292.448,E2 -19292.448} C_VEL
LIN {X 0,Y 241.793,Z 486.364,A -85,B 0,C 180,E1 -19295.544,E2 -19295.544} C_VEL
LIN {X 0,Y 241.952,Z 486.348,A -85,B 0,C 180,E1 -19298.346,E2 -19298.346} C_VEL
LIN {X 0,Y 241.936,Z 486.346,A -85,B 0,C 180,E1 -19301.924,E2 -19301.924} C_VEL
LIN {X 0,Y 241.937,Z 486.348,A -85,B 0,C 180,E1 -19306.571,E2 -19306.571} C_VEL
LIN {X 0,Y 241.976,Z 486.342,A -85,B 0,C 180,E1 -19310.285,E2 -19310.285} C_VEL
LIN {X 0,Y 242.04,Z 486.335,A -85,B 0,C 180,E1 -19314.498,E2 -19314.498} C_VEL
LIN {X 0,Y 241.98,Z 486.34,A -85,B 0,C 180,E1 -19318.48,E2 -19318.48} C_VEL
LIN {X 0,Y 242.012,Z 486.34,A -85,B 0,C 180,E1 -19322.313,E2 -19322.313} C_VEL
LIN {X 0,Y 242.062,Z 486.334,A -85,B 0,C 180,E1 -19326.016,E2 -19326.016} C_VEL
LIN {X 0,Y 242.042,Z 486.332,A -85,B 0,C 180,E1 -19329.608,E2 -19329.608} C_VEL
LIN {X 0,Y 242.167,Z 486.317,A -85,B 0,C 180,E1 -19333.278,E2 -19333.278} C_VEL
LIN {X 0,Y 242.191,Z 486.316,A -85,B 0,C 180,E1 -19338.28,E2 -19338.28} C_VEL
LIN {X 0,Y 242.44,Z 486.285,A -85,B 0,C 180,E1 -19341.666,E2 -19341.666} C_VEL
LIN {X 0,Y 242.265,Z 486.303,A -85,B 0,C 180,E1 -19345.007,E2 -19345.007} C_VEL
LIN {X 0,Y 242.641,Z 486.26,A -85,B 0,C 180,E1 -19348.34,E2 -19348.34} C_VEL
LIN {X 0,Y 242.64,Z 486.26,A -85,B 0,C 180,E1 -19351.66,E2 -19351.66} C_VEL
LIN {X 0,Y 242.413,Z 486.287,A -85,B 0,C 180,E1 -19356.659,E2 -19356.659} C_VEL
LIN {X 0,Y 242.272,Z 486.307,A -85,B 0,C 180,E1 -19360.024,E2 -19360.024} C_VEL
LIN {X 0,Y 242.172,Z 486.316,A -85,B 0,C 180,E1 -19365.141,E2 -19365.141} C_VEL
LIN {X 0,Y 242.078,Z 486.329,A -85,B 0,C 180,E1 -19368.624,E2 -19368.624} C_VEL
LIN {X 0,Y 242.016,Z 486.336,A -85,B 0,C 180,E1 -19372.18,E2 -19372.18} C_VEL
LIN {X 0,Y 242.07,Z 486.333,A -85,B 0,C 180,E1 -19375.838,E2 -19375.838} C_VEL
LIN {X 0,Y 242.033,Z 486.336,A -85,B 0,C 180,E1 -19379.58,E2 -19379.58} C_VEL
LIN {X 0,Y 241.995,Z 486.34,A -85,B 0,C 180,E1 -19383.49,E2 -19383.49} C_VEL
LIN {X 0,Y 242.006,Z 486.34,A -85,B 0,C 180,E1 -19387.579,E2 -19387.579} C_VEL
LIN {X 0,Y 241.946,Z 486.348,A -85,B 0,C 180,E1 -19391.921,E2 -19391.921} C_VEL
LIN {X 0,Y 241.937,Z 486.345,A -85,B 0,C 180,E1 -19396.571,E2 -19396.571} C_VEL
LIN {X 0,Y 241.954,Z 486.344,A -85,B 0,C 180,E1 -19400.28,E2 -19400.28} C_VEL
LIN {X 0,Y 241.882,Z 486.352,A -85,B 0,C 180,E1 -19404.445,E2 -19404.445} C_VEL
LIN {X 0,Y 241.545,Z 486.394,A -85,B 0,C 180,E1 -19408.417,E2 -19408.417} C_VEL
LIN {X 0,Y 241.081,Z 486.453,A -85,B 0,C 180,E1 -19412.196,E2 -19412.196} C_VEL
LIN {X 0,Y 240.541,Z 486.526,A -85,B 0,C 180,E1 -19417.053,E2 -19417.053} C_VEL
LIN {X 0,Y 242.823,Z 499.876,A -85,B 0,C 180,E1 -19418.171,E2 -19418.171} C_VEL
LIN {X 0,Y 244.919,Z 512.069,A -85,B 0,C 180,E1 -19419.462,E2 -19419.462} C_VEL
LIN {X 0,Y 246.154,Z 519.746,A -85,B 0,C 180,E1 -19420.423,E2 -19420.423} C_VEL
LIN {X 0,Y 244.877,Z 532.552,A -85,B 0,C 180,E1 -19422.245,E2 -19422.245} C_VEL
LIN {X 0,Y 243.672,Z 543.026,A -85,B 0,C 180,E1 -19424.097,E2 -19424.097} C_VEL
LIN {X 0,Y 242.515,Z 552.706,A -85,B 0,C 180,E1 -19426.167,E2 -19426.167} C_VEL
LIN {X 0,Y 241.542,Z 562.292,A -85,B 0,C 180,E1 -19428.673,E2 -19428.673} C_VEL
LIN {X 0,Y 240.833,Z 570.17,A -85,B 0,C 180,E1 -19431.187,E2 -19431.187} C_VEL
LIN {X 0,Y 240.296,Z 577.084,A -85,B 0,C 180,E1 -19433.939,E2 -19433.939} C_VEL
LIN {X 0,Y 240.156,Z 582.466,A -85,B 0,C 180,E1 -19436.644,E2 -19436.644} C_VEL
LIN {X 0,Y 240.07,Z 586.331,A -85,B 0,C 180,E1 -19439.161,E2 -19439.161} C_VEL
LIN {X 0,Y 240.228,Z 589.238,A -85,B 0,C 180,E1 -19441.676,E2 -19441.676} C_VEL
LIN {X 0,Y 240.516,Z 590.687,A -85,B 0,C 180,E1 -19443.35,E2 -19443.35} C_VEL
LIN {X 0,Y 240.856,Z 591.746,A -85,B 0,C 180,E1 -19445.022,E2 -19445.022} C_VEL
LIN {X 0,Y 241.845,Z 592.685,A -85,B 0,C 180,E1 -19448.354,E2 -19448.354} C_VEL
LIN {X 0,Y 243.794,Z 592.163,A -85,B 0,C 180,E1 -19451.642,E2 -19451.642} C_VEL
LIN {X 0,Y 244.803,Z 591.374,A -85,B 0,C 180,E1 -19453.277,E2 -19453.277} C_VEL
LIN {X 0,Y 247.919,Z 588.617,A -85,B 0,C 180,E1 -19456.468,E2 -19456.468} C_VEL
LIN {X 0,Y 250.593,Z 585.585,A -85,B 0,C 180,E1 -19458.815,E2 -19458.815} C_VEL
LIN {X 0,Y 255.011,Z 580.149,A -85,B 0,C 180,E1 -19461.842,E2 -19461.842} C_VEL
LIN {X 0,Y 260.167,Z 572.909,A -85,B 0,C 180,E1 -19464.753,E2 -19464.753} C_VEL
LIN {X 0,Y 265.384,Z 564.876,A -85,B 0,C 180,E1 -19467.182,E2 -19467.182} C_VEL
LIN {X 0,Y 270.257,Z 556.632,A -85,B 0,C 180,E1 -19469.182,E2 -19469.182} C_VEL
LIN {X 0,Y 271.848,Z 553.592,A -85,B 0,C 180,E1 -19469.846,E2 -19469.846} C_VEL
LIN {X 0,Y 272.21,Z 549.149,A -85,B 0,C 180,E1 -19471.569,E2 -19471.569} C_VEL
LIN {X 0,Y 272.08,Z 544.355,A -85,B 0,C 180,E1 -19473.755,E2 -19473.755} C_VEL
LIN {X 0,Y 271.791,Z 541.076,A -85,B 0,C 180,E1 -19475.523,E2 -19475.523} C_VEL
LIN {X 0,Y 271.209,Z 538.284,A -85,B 0,C 180,E1 -19477.567,E2 -19477.567} C_VEL
LIN {X 0,Y 270.286,Z 535.82,A -85,B 0,C 180,E1 -19480.832,E2 -19480.832} C_VEL
LIN {X 0,Y 269.803,Z 535.953,A -85,B 0,C 180,E1 -19482.08,E2 -19482.08} C_VEL
LIN {X 0,Y 268.876,Z 537.153,A -85,B 0,C 180,E1 -19483.304,E2 -19483.304} C_VEL
LIN {X 0,Y 266.434,Z 542.21,A -85,B 0,C 180,E1 -19486.55,E2 -19486.55} C_VEL
LIN {X 0,Y 266.308,Z 543.2,A -85,B 0,C 180,E1 -19487.395,E2 -19487.395} C_VEL
LIN {X 0,Y 266.445,Z 544.689,A -85,B 0,C 180,E1 -19488.744,E2 -19488.744} C_VEL
LIN {X 0,Y 266.499,Z 546.378,A -85,B 0,C 180,E1 -19489.887,E2 -19489.887} C_VEL
LIN {X 0,Y 266.017,Z 550.466,A -85,B 0,C 180,E1 -19491.713,E2 -19491.713} C_VEL
LIN {X 0,Y 265.278,Z 554.383,A -85,B 0,C 180,E1 -19493.086,E2 -19493.086} C_VEL
LIN {X 0,Y 262.844,Z 563.581,A -85,B 0,C 180,E1 -19495.84,E2 -19495.84} C_VEL
LIN {X 0,Y 259.585,Z 573.295,A -85,B 0,C 180,E1 -19498.589,E2 -19498.589} C_VEL
LIN {X 0,Y 256.693,Z 580.033,A -85,B 0,C 180,E1 -19500.474,E2 -19500.474} C_VEL
LIN {X 0,Y 252.289,Z 587.613,A -85,B 0,C 180,E1 -19502.636,E2 -19502.636} C_VEL
LIN {X 0,Y 247.933,Z 594.259,A -85,B 0,C 180,E1 -19504.837,E2 -19504.837} C_VEL
LIN {X 0,Y 242.91,Z 601.496,A -85,B 0,C 180,E1 -19507.906,E2 -19507.906} C_VEL
LIN {X 0,Y 239.169,Z 607.111,A -85,B 0,C 180,E1 -19511.141,E2 -19511.141} C_VEL
LIN {X 0,Y 236.098,Z 611.218,A -85,B 0,C 180,E1 -19514.46,E2 -19514.46} C_VEL
LIN {X 0,Y 234.166,Z 613.907,A -85,B 0,C 180,E1 -19517.872,E2 -19517.872} C_VEL
LIN {X 0,Y 233.177,Z 615.19,A -85,B 0,C 180,E1 -19521.332,E2 -19521.332} C_VEL
LIN {X 0,Y 233.008,Z 614.973,A -85,B 0,C 180,E1 -19524.808,E2 -19524.808} C_VEL
LIN {X 0,Y 233.42,Z 613.293,A -85,B 0,C 180,E1 -19528.275,E2 -19528.275} C_VEL
LIN {X 0,Y 233.63,Z 612.641,A -85,B 0,C 180,E1 -19529.354,E2 -19529.354} C_VEL
LIN {X 0,Y 233.316,Z 614.741,A -85,B 0,C 180,E1 -19531.726,E2 -19531.726} C_VEL
LIN {X 0,Y 232.968,Z 616.407,A -85,B 0,C 180,E1 -19535.192,E2 -19535.192} C_VEL
LIN {X 0,Y 233.169,Z 616.581,A -85,B 0,C 180,E1 -19538.668,E2 -19538.668} C_VEL
LIN {X 0,Y 234.178,Z 615.284,A -85,B 0,C 180,E1 -19542.127,E2 -19542.127} C_VEL
LIN {X 0,Y 236.094,Z 612.608,A -85,B 0,C 180,E1 -19545.54,E2 -19545.54} C_VEL
LIN {X 0,Y 239.093,Z 608.521,A -85,B 0,C 180,E1 -19548.865,E2 -19548.865} C_VEL
LIN {X 0,Y 242.078,Z 604.082,A -85,B 0,C 180,E1 -19551.53,E2 -19551.53} C_VEL
LIN {X 0,Y 246.512,Z 597.742,A -85,B 0,C 180,E1 -19554.418,E2 -19554.418} C_VEL
LIN {X 0,Y 251.489,Z 590.389,A -85,B 0,C 180,E1 -19557.008,E2 -19557.008} C_VEL
LIN {X 0,Y 256.93,Z 581.657,A -85,B 0,C 180,E1 -19559.497,E2 -19559.497} C_VEL
LIN {X 0,Y 259.34,Z 576.323,A -85,B 0,C 180,E1 -19560.99,E2 -19560.99} C_VEL
LIN {X 0,Y 261.703,Z 568.474,A -85,B 0,C 180,E1 -19563.392,E2 -19563.392} C_VEL
LIN {X 0,Y 263.233,Z 560.831,A -85,B 0,C 180,E1 -19565.971,E2 -19565.971} C_VEL
LIN {X 0,Y 264.172,Z 554.643,A -85,B 0,C 180,E1 -19568.39,E2 -19568.39} C_VEL
LIN {X 0,Y 264.492,Z 552.002,A -85,B 0,C 180,E1 -19569.622,E2 -19569.622} C_VEL
LIN {X 0,Y 264.565,Z 548.82,A -85,B 0,C 180,E1 -19571.614,E2 -19571.614} C_VEL
LIN {X 0,Y 264.707,Z 546.072,A -85,B 0,C 180,E1 -19574.205,E2 -19574.205} C_VEL
LIN {X 0,Y 264.816,Z 544.995,A -85,B 0,C 180,E1 -19576.369,E2 -19576.369} C_VEL
LIN {X 0,Y 264.859,Z 545.101,A -85,B 0,C 180,E1 -19578.443,E2 -19578.443} C_VEL
LIN {X 0,Y 265.234,Z 545.794,A -85,B 0,C 180,E1 -19580.511,E2 -19580.511} C_VEL
LIN {X 0,Y 266.039,Z 547.968,A -85,B 0,C 180,E1 -19583.382,E2 -19583.382} C_VEL
LIN {X 0,Y 266.351,Z 550.498,A -85,B 0,C 180,E1 -19585.291,E2 -19585.291} C_VEL
LIN {X 0,Y 266.532,Z 554.304,A -85,B 0,C 180,E1 -19587.543,E2 -19587.543} C_VEL
LIN {X 0,Y 266.283,Z 558.172,A -85,B 0,C 180,E1 -19589.417,E2 -19589.417} C_VEL
LIN {X 0,Y 265.77,Z 559.493,A -85,B 0,C 180,E1 -19589.839,E2 -19589.839} C_VEL
LIN {X 0,Y 260.609,Z 567.419,A -85,B 0,C 180,E1 -19591.84,E2 -19591.84} C_VEL
LIN {X 0,Y 254.334,Z 576.035,A -85,B 0,C 180,E1 -19594.64,E2 -19594.64} C_VEL
LIN {X 0,Y 250.127,Z 581.242,A -85,B 0,C 180,E1 -19596.836,E2 -19596.836} C_VEL
LIN {X 0,Y 245.329,Z 586.632,A -85,B 0,C 180,E1 -19599.894,E2 -19599.894} C_VEL
LIN {X 0,Y 241.395,Z 590.505,A -85,B 0,C 180,E1 -19603.074,E2 -19603.074} C_VEL
LIN {X 0,Y 239.638,Z 591.889,A -85,B 0,C 180,E1 -19604.696,E2 -19604.696} C_VEL
LIN {X 0,Y 237.019,Z 593.542,A -85,B 0,C 180,E1 -19608.021,E2 -19608.021} C_VEL
LIN {X 0,Y 234.913,Z 593.824,A -85,B 0,C 180,E1 -19611.397,E2 -19611.397} C_VEL
LIN {X 0,Y 233.882,Z 592.598,A -85,B 0,C 180,E1 -19614.828,E2 -19614.828} C_VEL
LIN {X 0,Y 233.191,Z 589.91,A -85,B 0,C 180,E1 -19618.273,E2 -19618.273} C_VEL
LIN {X 0,Y 233.023,Z 586.838,A -85,B 0,C 180,E1 -19620.864,E2 -19620.864} C_VEL
LIN {X 0,Y 233.081,Z 582.801,A -85,B 0,C 180,E1 -19623.458,E2 -19623.458} C_VEL
LIN {X 0,Y 233.279,Z 577.427,A -85,B 0,C 180,E1 -19626.176,E2 -19626.176} C_VEL
LIN {X 0,Y 233.732,Z 571.397,A -85,B 0,C 180,E1 -19628.647,E2 -19628.647} C_VEL
LIN {X 0,Y 234.406,Z 563.651,A -85,B 0,C 180,E1 -19631.238,E2 -19631.238} C_VEL
LIN {X 0,Y 235.371,Z 554.122,A -85,B 0,C 180,E1 -19633.821,E2 -19633.821} C_VEL
LIN {X 0,Y 236.643,Z 543.556,A -85,B 0,C 180,E1 -19636.167,E2 -19636.167} C_VEL
LIN {X 0,Y 238.012,Z 531.725,A -85,B 0,C 180,E1 -19638.285,E2 -19638.285} C_VEL
LIN {X 0,Y 239.176,Z 520.236,A -85,B 0,C 180,E1 -19639.963,E2 -19639.963} C_VEL
LIN {X 0,Y 236.927,Z 507.509,A -85,B 0,C 180,E1 -19641.53,E2 -19641.53} C_VEL
LIN {X 0,Y 234.611,Z 494.496,A -85,B 0,C 180,E1 -19642.825,E2 -19642.825} C_VEL
LIN {X 0,Y 233.541,Z 487.399,A -85,B 0,C 180,E1 -19643.441,E2 -19643.441} C_VEL
LIN {X 0,Y 233.853,Z 487.357,A -85,B 0,C 180,E1 -19646.795,E2 -19646.795} C_VEL
LIN {X 0,Y 234.259,Z 487.303,A -85,B 0,C 180,E1 -19650.666,E2 -19650.666} C_VEL
LIN {X 0,Y 234.639,Z 487.256,A -85,B 0,C 180,E1 -19654.688,E2 -19654.688} C_VEL
LIN {X 0,Y 234.889,Z 487.224,A -85,B 0,C 180,E1 -19658.928,E2 -19658.928} C_VEL
LIN {X 0,Y 234.89,Z 487.223,A -85,B 0,C 180,E1 -19663.486,E2 -19663.486} C_VEL
LIN {X 0,Y 234.89,Z 487.226,A -85,B 0,C 180,E1 -19666.514,E2 -19666.514} C_VEL
LIN {X 0,Y 234.958,Z 487.213,A -85,B 0,C 180,E1 -19671.086,E2 -19671.086} C_VEL
LIN {X 0,Y 234.964,Z 487.215,A -85,B 0,C 180,E1 -19675.368,E2 -19675.368} C_VEL
LIN {X 0,Y 234.972,Z 487.214,A -85,B 0,C 180,E1 -19680.158,E2 -19680.158} C_VEL
LIN {X 0,Y 234.998,Z 487.212,A -85,B 0,C 180,E1 -19683.794,E2 -19683.794} C_VEL
LIN {X 0,Y 235.016,Z 487.206,A -85,B 0,C 180,E1 -19688.97,E2 -19688.97} C_VEL
LIN {X 0,Y 235.101,Z 487.198,A -85,B 0,C 180,E1 -19693.059,E2 -19693.059} C_VEL
LIN {X 0,Y 235.152,Z 487.191,A -85,B 0,C 180,E1 -19697.924,E2 -19697.924} C_VEL
LIN {X 0,Y 235.395,Z 487.162,A -85,B 0,C 180,E1 -19701.415,E2 -19701.415} C_VEL
LIN {X 0,Y 235.411,Z 487.159,A -85,B 0,C 180,E1 -19703.142,E2 -19703.142} C_VEL
LIN {X 0,Y 235.601,Z 487.138,A -85,B 0,C 180,E1 -19708.291,E2 -19708.291} C_VEL
LIN {X 0,Y 235.599,Z 487.138,A -85,B 0,C 180,E1 -19711.709,E2 -19711.709} C_VEL
LIN {X 0,Y 235.364,Z 487.164,A -85,B 0,C 180,E1 -19716.86,E2 -19716.86} C_VEL
LIN {X 0,Y 235.219,Z 487.184,A -85,B 0,C 180,E1 -19720.327,E2 -19720.327} C_VEL
LIN {X 0,Y 235.118,Z 487.196,A -85,B 0,C 180,E1 -19725.606,E2 -19725.606} C_VEL
LIN {X 0,Y 235.013,Z 487.209,A -85,B 0,C 180,E1 -19729.205,E2 -19729.205} C_VEL
LIN {X 0,Y 234.964,Z 487.212,A -85,B 0,C 180,E1 -19732.883,E2 -19732.883} C_VEL
LIN {X 0,Y 234.973,Z 487.214,A -85,B 0,C 180,E1 -19736.657,E2 -19736.657} C_VEL
LIN {X 0,Y 234.935,Z 487.215,A -85,B 0,C 180,E1 -19740.567,E2 -19740.567} C_VEL
LIN {X 0,Y 234.964,Z 487.215,A -85,B 0,C 180,E1 -19744.632,E2 -19744.632} C_VEL
LIN {X 0,Y 234.945,Z 487.215,A -85,B 0,C 180,E1 -19748.944,E2 -19748.944} C_VEL
LIN {X 0,Y 234.89,Z 487.226,A -85,B 0,C 180,E1 -19753.486,E2 -19753.486} C_VEL
LIN {X 0,Y 234.89,Z 487.223,A -85,B 0,C 180,E1 -19756.514,E2 -19756.514} C_VEL
LIN {X 0,Y 234.92,Z 487.22,A -85,B 0,C 180,E1 -19761.078,E2 -19761.078} C_VEL
LIN {X 0,Y 234.854,Z 487.231,A -85,B 0,C 180,E1 -19763.899,E2 -19763.899} C_VEL
LIN {X 0,Y 234.62,Z 487.257,A -85,B 0,C 180,E1 -19767.371,E2 -19767.371} C_VEL
LIN {X 0,Y 234.147,Z 487.318,A -85,B 0,C 180,E1 -19771.298,E2 -19771.298} C_VEL
LIN {X 0,Y 233.591,Z 487.388,A -85,B 0,C 180,E1 -19776.035,E2 -19776.035} C_VEL
LIN {X 0,Y 233.527,Z 487.398,A -85,B 0,C 180,E1 -19776.88,E2 -19776.88} C_VEL
LIN {X 0,Y 235.981,Z 501.863,A -85,B 0,C 180,E1 -19778.152,E2 -19778.152} C_VEL
LIN {X 0,Y 238.419,Z 515.971,A -85,B 0,C 180,E1 -19779.76,E2 -19779.76} C_VEL
LIN {X 0,Y 238.996,Z 519.457,A -85,B 0,C 180,E1 -19780.221,E2 -19780.221} C_VEL
LIN {X 0,Y 237.923,Z 531.296,A -85,B 0,C 180,E1 -19781.931,E2 -19781.931} C_VEL
LIN {X 0,Y 236.573,Z 543.084,A -85,B 0,C 180,E1 -19784.05,E2 -19784.05} C_VEL
LIN {X 0,Y 235.385,Z 552.835,A -85,B 0,C 180,E1 -19786.18,E2 -19786.18} C_VEL
LIN {X 0,Y 234.41,Z 562.479,A -85,B 0,C 180,E1 -19788.762,E2 -19788.762} C_VEL
LIN {X 0,Y 233.706,Z 570.397,A -85,B 0,C 180,E1 -19791.352,E2 -19791.352} C_VEL
LIN {X 0,Y 233.197,Z 576.933,A -85,B 0,C 180,E1 -19794.013,E2 -19794.013} C_VEL
LIN {X 0,Y 233.076,Z 581.974,A -85,B 0,C 180,E1 -19796.542,E2 -19796.542} C_VEL
LIN {X 0,Y 232.998,Z 586.075,A -85,B 0,C 180,E1 -19799.135,E2 -19799.135} C_VEL
LIN {X 0,Y 233.156,Z 589.201,A -85,B 0,C 180,E1 -19801.727,E2 -19801.727} C_VEL
LIN {X 0,Y 233.787,Z 591.92,A -85,B 0,C 180,E1 -19805.174,E2 -19805.174} C_VEL
LIN {X 0,Y 234.853,Z 593.194,A -85,B 0,C 180,E1 -19808.605,E2 -19808.605} C_VEL
LIN {X 0,Y 236.873,Z 592.932,A -85,B 0,C 180,E1 -19811.987,E2 -19811.987} C_VEL
LIN {X 0,Y 237.97,Z 592.299,A -85,B 0,C 180,E1 -19813.666,E2 -19813.666} C_VEL
LIN {X 0,Y 241.252,Z 589.894,A -85,B 0,C 180,E1 -19816.936,E2 -19816.936} C_VEL
LIN {X 0,Y 244.058,Z 587.165,A -85,B 0,C 180,E1 -19819.339,E2 -19819.339} C_VEL
LIN {X 0,Y 248.663,Z 582.069,A -85,B 0,C 180,E1 -19822.43,E2 -19822.43} C_VEL
LIN {X 0,Y 252.62,Z 577.196,A -85,B 0,C 180,E1 -19824.664,E2 -19824.664} C_VEL
LIN {X 0,Y 257.869,Z 570.187,A -85,B 0,C 180,E1 -19827.162,E2 -19827.162} C_VEL
LIN {X 0,Y 263.631,Z 561.502,A -85,B 0,C 180,E1 -19829.55,E2 -19829.55} C_VEL
LIN {X 0,Y 266.572,Z 556.791,A -85,B 0,C 180,E1 -19830.643,E2 -19830.643} C_VEL
LIN {X 0,Y 267.134,Z 552.145,A -85,B 0,C 180,E1 -19832.66,E2 -19832.66} C_VEL
LIN {X 0,Y 267.227,Z 547.023,A -85,B 0,C 180,E1 -19835.383,E2 -19835.383} C_VEL
LIN {X 0,Y 266.89,Z 543.805,A -85,B 0,C 180,E1 -19837.815,E2 -19837.815} C_VEL
LIN {X 0,Y 266.259,Z 541.519,A -85,B 0,C 180,E1 -19841.291,E2 -19841.291} C_VEL
LIN {X 0,Y 266.25,Z 541.045,A -85,B 0,C 180,E1 -19843.338,E2 -19843.338} C_VEL
LIN {X 0,Y 266.292,Z 541.172,A -85,B 0,C 180,E1 -19844.554,E2 -19844.554} C_VEL
LIN {X 0,Y 266.287,Z 542.5,A -85,B 0,C 180,E1 -19846.669,E2 -19846.669} C_VEL
LIN {X 0,Y 266.308,Z 543.2,A -85,B 0,C 180,E1 -19847.395,E2 -19847.395} C_VEL
LIN {X 0,Y 266.173,Z 544.35,A -85,B 0,C 180,E1 -19848.204,E2 -19848.204} C_VEL
LIN {X 0,Y 265.378,Z 547.061,A -85,B 0,C 180,E1 -19849.327,E2 -19849.327} C_VEL
LIN {X 0,Y 263.994,Z 550.482,A -85,B 0,C 180,E1 -19850.349,E2 -19850.349} C_VEL
LIN {X 0,Y 261.7,Z 555.684,A -85,B 0,C 180,E1 -19851.668,E2 -19851.668} C_VEL
LIN {X 0,Y 259.769,Z 560.538,A -85,B 0,C 180,E1 -19853.058,E2 -19853.058} C_VEL
LIN {X 0,Y 256.774,Z 569.138,A -85,B 0,C 180,E1 -19855.762,E2 -19855.762} C_VEL
LIN {X 0,Y 252.833,Z 578.449,A -85,B 0,C 180,E1 -19858.588,E2 -19858.588} C_VEL
LIN {X 0,Y 248.567,Z 585.867,A -85,B 0,C 180,E1 -19860.809,E2 -19860.809} C_VEL
LIN {X 0,Y 243.085,Z 593.607,A -85,B 0,C 180,E1 -19863.376,E2 -19863.376} C_VEL
LIN {X 0,Y 237.677,Z 600.794,A -85,B 0,C 180,E1 -19866.471,E2 -19866.471} C_VEL
LIN {X 0,Y 233.366,Z 606.406,A -85,B 0,C 180,E1 -19869.737,E2 -19869.737} C_VEL
LIN {X 0,Y 230.801,Z 609.606,A -85,B 0,C 180,E1 -19872.272,E2 -19872.272} C_VEL
LIN {X 0,Y 228.034,Z 612.701,A -85,B 0,C 180,E1 -19875.726,E2 -19875.726} C_VEL
LIN {X 0,Y 226.565,Z 614.362,A -85,B 0,C 180,E1 -19879.274,E2 -19879.274} C_VEL
LIN {X 0,Y 225.965,Z 614.637,A -85,B 0,C 180,E1 -19882.853,E2 -19882.853} C_VEL
LIN {X 0,Y 225.95,Z 614.249,A -85,B 0,C 180,E1 -19884.646,E2 -19884.646} C_VEL
LIN {X 0,Y 226.4,Z 612.285,A -85,B 0,C 180,E1 -19888.221,E2 -19888.221} C_VEL
LIN {X 0,Y 226.614,Z 611.496,A -85,B 0,C 180,E1 -19889.334,E2 -19889.334} C_VEL
LIN {X 0,Y 226.285,Z 613.768,A -85,B 0,C 180,E1 -19891.78,E2 -19891.78} C_VEL
LIN {X 0,Y 225.922,Z 615.651,A -85,B 0,C 180,E1 -19895.355,E2 -19895.355} C_VEL
LIN {X 0,Y 226.153,Z 616.056,A -85,B 0,C 180,E1 -19898.939,E2 -19898.939} C_VEL
LIN {X 0,Y 227.195,Z 615.063,A -85,B 0,C 180,E1 -19902.506,E2 -19902.506} C_VEL
LIN {X 0,Y 229.25,Z 612.694,A -85,B 0,C 180,E1 -19906.016,E2 -19906.016} C_VEL
LIN {X 0,Y 232.384,Z 608.934,A -85,B 0,C 180,E1 -19909.431,E2 -19909.431} C_VEL
LIN {X 0,Y 236.368,Z 603.762,A -85,B 0,C 180,E1 -19912.739,E2 -19912.739} C_VEL
LIN {X 0,Y 240.147,Z 598.882,A -85,B 0,C 180,E1 -19915.11,E2 -19915.11} C_VEL
LIN {X 0,Y 246.129,Z 590.933,A -85,B 0,C 180,E1 -19918.109,E2 -19918.109} C_VEL
LIN {X 0,Y 251.034,Z 583.774,A -85,B 0,C 180,E1 -19920.261,E2 -19920.261} C_VEL
LIN {X 0,Y 253.654,Z 578.785,A -85,B 0,C 180,E1 -19921.765,E2 -19921.765} C_VEL
LIN {X 0,Y 256.108,Z 572.06,A -85,B 0,C 180,E1 -19923.977,E2 -19923.977} C_VEL
LIN {X 0,Y 257.899,Z 565.532,A -85,B 0,C 180,E1 -19926.319,E2 -19926.319} C_VEL
LIN {X 0,Y 259.164,Z 560.004,A -85,B 0,C 180,E1 -19928.588,E2 -19928.588} C_VEL
LIN {X 0,Y 259.898,Z 556.274,A -85,B 0,C 180,E1 -19930.466,E2 -19930.466} C_VEL
LIN {X 0,Y 260.123,Z 553.503,A -85,B 0,C 180,E1 -19932.489,E2 -19932.489} C_VEL
LIN {X 0,Y 260.388,Z 551.505,A -85,B 0,C 180,E1 -19934.568,E2 -19934.568} C_VEL
LIN {X 0,Y 260.504,Z 550.615,A -85,B 0,C 180,E1 -19936.754,E2 -19936.754} C_VEL
LIN {X 0,Y 260.63,Z 551.068,A -85,B 0,C 180,E1 -19939.672,E2 -19939.672} C_VEL
